LIN {X 0,Y 388.393,Z 704.087,A -85,B 0,C 180,E1 -23559.854,E2 -23559.854} C_VEL
LIN {X 0,Y 400.252,Z 573.446,A -85,B 0,C 180,E1 -23561.917,E2 -23561.917} C_VEL
LIN {X 0,Y 395.946,Z 563.972,A -85,B 0,C 180,E1 -23564.361,E2 -23564.361} C_VEL
LIN {X 0,Y 391.725,Z 556.337,A -85,B 0,C 180,E1 -23567.094,E2 -23567.094} C_VEL
LIN {X 0,Y 388.594,Z 550.898,A -85,B 0,C 180,E1 -23569.548,E2 -23569.548} C_VEL
LIN {X 0,Y 386.254,Z 546.876,A -85,B 0,C 180,E1 -23571.815,E2 -23571.815} C_VEL
LIN {X 0,Y 383.997,Z 542.829,A -85,B 0,C 180,E1 -23574.771,E2 -23574.771} C_VEL
LIN {X 0,Y 382.142,Z 538.278,A -85,B 0,C 180,E1 -23581.349,E2 -23581.349} C_VEL
LIN {X 0,Y 384.382,Z 543.419,A -85,B 0,C 180,E1 -23588.226,E2 -23588.226} C_VEL
LIN {X 0,Y 387.171,Z 548.383,A -85,B 0,C 180,E1 -23591.546,E2 -23591.546} C_VEL
LIN {X 0,Y 389.894,Z 553.166,A -85,B 0,C 180,E1 -23593.949,E2 -23593.949} C_VEL
LIN {X 0,Y 393.621,Z 559.599,A -85,B 0,C 180,E1 -23596.605,E2 -23596.605} C_VEL
LIN {X 0,Y 398.687,Z 569.021,A -85,B 0,C 180,E1 -23599.599,E2 -23599.599} C_VEL
LIN {X 0,Y 400.284,Z 572.367,A -85,B 0,C 180,E1 -23600.456,E2 -23600.456} C_VEL
LIN {X 0,Y 384.057,Z 748.302,A -85,B 0,C 180,E1 -23603.233,E2 -23603.233} C_VEL
LIN {X 0,Y 380.026,Z 774.745,A -85,B 0,C 180,E1 -23603.787,E2 -23603.787} C_VEL
LIN {X 0,Y 375.691,Z 795.491,A -85,B 0,C 180,E1 -23604.362,E2 -23604.362} C_VEL
LIN {X 0,Y 369.224,Z 820.189,A -85,B 0,C 180,E1 -23605.244,E2 -23605.244} C_VEL
LIN {X 0,Y 362.641,Z 840.771,A -85,B 0,C 180,E1 -23606.178,E2 -23606.178} C_VEL
LIN {X 0,Y 354.698,Z 862.408,A -85,B 0,C 180,E1 -23607.379,E2 -23607.379} C_VEL
LIN {X 0,Y 345.362,Z 883.966,A -85,B 0,C 180,E1 -23608.861,E2 -23608.861} C_VEL
LIN {X 0,Y 335.768,Z 903.879,A -85,B 0,C 180,E1 -23610.523,E2 -23610.523} C_VEL
LIN {X 0,Y 325.015,Z 923.613,A -85,B 0,C 180,E1 -23612.548,E2 -23612.548} C_VEL
LIN {X 0,Y 314.859,Z 940.708,A -85,B 0,C 180,E1 -23614.664,E2 -23614.664} C_VEL
LIN {X 0,Y 303.227,Z 958.602,A -85,B 0,C 180,E1 -23617.373,E2 -23617.373} C_VEL
LIN {X 0,Y 292.874,Z 973.436,A -85,B 0,C 180,E1 -23620.115,E2 -23620.115} C_VEL
LIN {X 0,Y 281.008,Z 989.437,A -85,B 0,C 180,E1 -23623.754,E2 -23623.754} C_VEL
LIN {X 0,Y 271.257,Z 1001.963,A -85,B 0,C 180,E1 -23627.293,E2 -23627.293} C_VEL
LIN {X 0,Y 261.14,Z 1014.647,A -85,B 0,C 180,E1 -23631.715,E2 -23631.715} C_VEL
LIN {X 0,Y 252.983,Z 1024.7,A -85,B 0,C 180,E1 -23636.132,E2 -23636.132} C_VEL
LIN {X 0,Y 245.579,Z 1034.158,A -85,B 0,C 180,E1 -23641.286,E2 -23641.286} C_VEL
LIN {X 0,Y 239.901,Z 1041.714,A -85,B 0,C 180,E1 -23646.675,E2 -23646.675} C_VEL
LIN {X 0,Y 235.924,Z 1047.812,A -85,B 0,C 180,E1 -23652.233,E2 -23652.233} C_VEL
LIN {X 0,Y 233.421,Z 1052.417,A -85,B 0,C 180,E1 -23658.135,E2 -23658.135} C_VEL
LIN {X 0,Y 232.411,Z 1055.085,A -85,B 0,C 180,E1 -23663.081,E2 -23663.081} C_VEL
LIN {X 0,Y 232.071,Z 1056.714,A -85,B 0,C 180,E1 -23668.025,E2 -23668.025} C_VEL
LIN {X 0,Y 232.018,Z 1057.307,A -85,B 0,C 180,E1 -23673.212,E2 -23673.212} C_VEL
LIN {X 0,Y 232.196,Z 1056.634,A -85,B 0,C 180,E1 -23678.419,E2 -23678.419} C_VEL
LIN {X 0,Y 232.853,Z 1054.948,A -85,B 0,C 180,E1 -23683.408,E2 -23683.408} C_VEL
LIN {X 0,Y 234.592,Z 1051.893,A -85,B 0,C 180,E1 -23688.901,E2 -23688.901} C_VEL
LIN {X 0,Y 238.088,Z 1046.847,A -85,B 0,C 180,E1 -23694.888,E2 -23694.888} C_VEL
LIN {X 0,Y 242.615,Z 1041.161,A -85,B 0,C 180,E1 -23699.913,E2 -23699.913} C_VEL
LIN {X 0,Y 250.02,Z 1032.531,A -85,B 0,C 180,E1 -23705.725,E2 -23705.725} C_VEL
LIN {X 0,Y 257.882,Z 1023.616,A -85,B 0,C 180,E1 -23710.354,E2 -23710.354} C_VEL
LIN {X 0,Y 268.413,Z 1011.672,A -85,B 0,C 180,E1 -23715.246,E2 -23715.246} C_VEL
LIN {X 0,Y 278.302,Z 1000.135,A -85,B 0,C 180,E1 -23718.981,E2 -23718.981} C_VEL
LIN {X 0,Y 290.19,Z 985.74,A -85,B 0,C 180,E1 -23722.744,E2 -23722.744} C_VEL
LIN {X 0,Y 301.246,Z 971.426,A -85,B 0,C 180,E1 -23725.739,E2 -23725.739} C_VEL
LIN {X 0,Y 313.044,Z 955.275,A -85,B 0,C 180,E1 -23728.52,E2 -23728.52} C_VEL
LIN {X 0,Y 324.773,Z 937.569,A -85,B 0,C 180,E1 -23730.969,E2 -23730.969} C_VEL
LIN {X 0,Y 335.952,Z 919.34,A -85,B 0,C 180,E1 -23733.049,E2 -23733.049} C_VEL
LIN {X 0,Y 346.746,Z 899.544,A -85,B 0,C 180,E1 -23734.886,E2 -23734.886} C_VEL
LIN {X 0,Y 355.593,Z 881.622,A -85,B 0,C 180,E1 -23736.264,E2 -23736.264} C_VEL
LIN {X 0,Y 365.537,Z 858.721,A -85,B 0,C 180,E1 -23737.71,E2 -23737.71} C_VEL
LIN {X 0,Y 372.878,Z 839.111,A -85,B 0,C 180,E1 -23738.723,E2 -23738.723} C_VEL
LIN {X 0,Y 380.335,Z 815.96,A -85,B 0,C 180,E1 -23739.694,E2 -23739.694} C_VEL
LIN {X 0,Y 386.25,Z 793.125,A -85,B 0,C 180,E1 -23740.44,E2 -23740.44} C_VEL
LIN {X 0,Y 391.244,Z 769.089,A -85,B 0,C 180,E1 -23741.046,E2 -23741.046} C_VEL
LIN {X 0,Y 394.683,Z 744.791,A -85,B 0,C 180,E1 -23741.5,E2 -23741.5} C_VEL
LIN {X 0,Y 410.348,Z 579.625,A -85,B 0,C 180,E1 -23744.054,E2 -23744.054} C_VEL
LIN {X 0,Y 405.942,Z 571.377,A -85,B 0,C 180,E1 -23746.83,E2 -23746.83} C_VEL
LIN {X 0,Y 402.359,Z 564.773,A -85,B 0,C 180,E1 -23749.621,E2 -23749.621} C_VEL
LIN {X 0,Y 400.956,Z 563.778,A -85,B 0,C 180,E1 -23750.779,E2 -23750.779} C_VEL
LIN {X 0,Y 397.256,Z 564.937,A -85,B 0,C 180,E1 -23754.266,E2 -23754.266} C_VEL
LIN {X 0,Y 396.971,Z 564.739,A -85,B 0,C 180,E1 -23754.666,E2 -23754.666} C_VEL
LIN {X 0,Y 395.189,Z 560.495,A -85,B 0,C 180,E1 -23760.87,E2 -23760.87} C_VEL
LIN {X 0,Y 397.102,Z 565.119,A -85,B 0,C 180,E1 -23767.233,E2 -23767.233} C_VEL
LIN {X 0,Y 399.583,Z 569.876,A -85,B 0,C 180,E1 -23770.38,E2 -23770.38} C_VEL
LIN {X 0,Y 402.269,Z 574.828,A -85,B 0,C 180,E1 -23772.854,E2 -23772.854} C_VEL
LIN {X 0,Y 405.294,Z 580.545,A -85,B 0,C 180,E1 -23775.123,E2 -23775.123} C_VEL
LIN {X 0,Y 407.597,Z 586.184,A -85,B 0,C 180,E1 -23776.699,E2 -23776.699} C_VEL
LIN {X 0,Y 391.12,Z 755.536,A -85,B 0,C 180,E1 -23779.285,E2 -23779.285} C_VEL
LIN {X 0,Y 386.856,Z 782.013,A -85,B 0,C 180,E1 -23779.789,E2 -23779.789} C_VEL
LIN {X 0,Y 382.071,Z 803.436,A -85,B 0,C 180,E1 -23780.299,E2 -23780.299} C_VEL
LIN {X 0,Y 375.038,Z 828.403,A -85,B 0,C 180,E1 -23781.071,E2 -23781.071} C_VEL
LIN {X 0,Y 367.984,Z 849.001,A -85,B 0,C 180,E1 -23781.886,E2 -23781.886} C_VEL
LIN {X 0,Y 359.022,Z 871.665,A -85,B 0,C 180,E1 -23783.007,E2 -23783.007} C_VEL
LIN {X 0,Y 349.433,Z 892.46,A -85,B 0,C 180,E1 -23784.304,E2 -23784.304} C_VEL
LIN {X 0,Y 338.891,Z 912.953,A -85,B 0,C 180,E1 -23785.856,E2 -23785.856} C_VEL
LIN {X 0,Y 327.505,Z 932.463,A -85,B 0,C 180,E1 -23787.701,E2 -23787.701} C_VEL
LIN {X 0,Y 316.516,Z 949.77,A -85,B 0,C 180,E1 -23789.687,E2 -23789.687} C_VEL
LIN {X 0,Y 303.867,Z 967.902,A -85,B 0,C 180,E1 -23792.256,E2 -23792.256} C_VEL
LIN {X 0,Y 293.193,Z 982.14,A -85,B 0,C 180,E1 -23794.725,E2 -23794.725} C_VEL
LIN {X 0,Y 280.683,Z 997.872,A -85,B 0,C 180,E1 -23798.068,E2 -23798.068} C_VEL
LIN {X 0,Y 269.384,Z 1011.222,A -85,B 0,C 180,E1 -23801.637,E2 -23801.637} C_VEL
LIN {X 0,Y 258.376,Z 1023.94,A -85,B 0,C 180,E1 -23805.847,E2 -23805.847} C_VEL
LIN {X 0,Y 248.504,Z 1034.966,A -85,B 0,C 180,E1 -23810.526,E2 -23810.526} C_VEL
LIN {X 0,Y 239.962,Z 1044.827,A -85,B 0,C 180,E1 -23815.769,E2 -23815.769} C_VEL
LIN {X 0,Y 233.287,Z 1052.746,A -85,B 0,C 180,E1 -23821.312,E2 -23821.312} C_VEL
LIN {X 0,Y 228.711,Z 1058.908,A -85,B 0,C 180,E1 -23826.83,E2 -23826.83} C_VEL
LIN {X 0,Y 225.515,Z 1064.125,A -85,B 0,C 180,E1 -23833.277,E2 -23833.277} C_VEL
LIN {X 0,Y 224.312,Z 1066.99,A -85,B 0,C 180,E1 -23838.428,E2 -23838.428} C_VEL
LIN {X 0,Y 223.979,Z 1068.777,A -85,B 0,C 180,E1 -23843.592,E2 -23843.592} C_VEL
LIN {X 0,Y 224.01,Z 1069.469,A -85,B 0,C 180,E1 -23848.721,E2 -23848.721} C_VEL
LIN {X 0,Y 223.991,Z 1069.015,A -85,B 0,C 180,E1 -23853.583,E2 -23853.583} C_VEL
LIN {X 0,Y 224.053,Z 1067.383,A -85,B 0,C 180,E1 -23858.727,E2 -23858.727} C_VEL
LIN {X 0,Y 224.71,Z 1064.64,A -85,B 0,C 180,E1 -23863.903,E2 -23863.903} C_VEL
LIN {X 0,Y 226.6,Z 1060.347,A -85,B 0,C 180,E1 -23869.594,E2 -23869.594} C_VEL
LIN {X 0,Y 230.424,Z 1053.913,A -85,B 0,C 180,E1 -23875.718,E2 -23875.718} C_VEL
LIN {X 0,Y 235.435,Z 1046.841,A -85,B 0,C 180,E1 -23880.923,E2 -23880.923} C_VEL
LIN {X 0,Y 243.47,Z 1036.499,A -85,B 0,C 180,E1 -23886.841,E2 -23886.841} C_VEL
LIN {X 0,Y 251.465,Z 1026.59,A -85,B 0,C 180,E1 -23891.304,E2 -23891.304} C_VEL
LIN {X 0,Y 262.304,Z 1013.248,A -85,B 0,C 180,E1 -23896.092,E2 -23896.092} C_VEL
LIN {X 0,Y 272.513,Z 1000.343,A -85,B 0,C 180,E1 -23899.776,E2 -23899.776} C_VEL
LIN {X 0,Y 284.845,Z 984.13,A -85,B 0,C 180,E1 -23903.5,E2 -23903.5} C_VEL
LIN {X 0,Y 295.676,Z 968.974,A -85,B 0,C 180,E1 -23906.294,E2 -23906.294} C_VEL
LIN {X 0,Y 307.858,Z 950.808,A -85,B 0,C 180,E1 -23909.031,E2 -23909.031} C_VEL
LIN {X 0,Y 318.866,Z 932.772,A -85,B 0,C 180,E1 -23911.217,E2 -23911.217} C_VEL
LIN {X 0,Y 329.909,Z 913.124,A -85,B 0,C 180,E1 -23913.179,E2 -23913.179} C_VEL
LIN {X 0,Y 340.246,Z 892.323,A -85,B 0,C 180,E1 -23914.84,E2 -23914.84} C_VEL
LIN {X 0,Y 349.638,Z 871.278,A -85,B 0,C 180,E1 -23916.224,E2 -23916.224} C_VEL
LIN {X 0,Y 358.028,Z 849.339,A -85,B 0,C 180,E1 -23917.37,E2 -23917.37} C_VEL
LIN {X 0,Y 364.543,Z 829.829,A -85,B 0,C 180,E1 -23918.195,E2 -23918.195} C_VEL
LIN {X 0,Y 371.552,Z 804.574,A -85,B 0,C 180,E1 -23919.038,E2 -23919.038} C_VEL
LIN {X 0,Y 376.275,Z 783.017,A -85,B 0,C 180,E1 -23919.588,E2 -23919.588} C_VEL
LIN {X 0,Y 380.395,Z 757.375,A -85,B 0,C 180,E1 -23920.106,E2 -23920.106} C_VEL
LIN {X 0,Y 387.874,Z 678.891,A -85,B 0,C 180,E1 -23921.359,E2 -23921.359} C_VEL
LIN {X 0,Y 397.206,Z 578.193,A -85,B 0,C 180,E1 -23922.946,E2 -23922.946} C_VEL
LIN {X 0,Y 393.989,Z 570.875,A -85,B 0,C 180,E1 -23924.884,E2 -23924.884} C_VEL
LIN {X 0,Y 389.653,Z 562.753,A -85,B 0,C 180,E1 -23927.853,E2 -23927.853} C_VEL
LIN {X 0,Y 387.019,Z 558.202,A -85,B 0,C 180,E1 -23930.032,E2 -23930.032} C_VEL
LIN {X 0,Y 384.996,Z 554.581,A -85,B 0,C 180,E1 -23932.088,E2 -23932.088} C_VEL
LIN {X 0,Y 382.923,Z 550.71,A -85,B 0,C 180,E1 -23934.907,E2 -23934.907} C_VEL
LIN {X 0,Y 381.159,Z 546.277,A -85,B 0,C 180,E1 -23941.353,E2 -23941.353} C_VEL
LIN {X 0,Y 383.252,Z 551.234,A -85,B 0,C 180,E1 -23948.024,E2 -23948.024} C_VEL
LIN {X 0,Y 385.89,Z 556.083,A -85,B 0,C 180,E1 -23951.282,E2 -23951.282} C_VEL
LIN {X 0,Y 388.626,Z 561.047,A -85,B 0,C 180,E1 -23953.768,E2 -23953.768} C_VEL
LIN {X 0,Y 392.071,Z 567.186,A -85,B 0,C 180,E1 -23956.292,E2 -23956.292} C_VEL
LIN {X 0,Y 397.023,Z 576.643,A -85,B 0,C 180,E1 -23959.302,E2 -23959.302} C_VEL
LIN {X 0,Y 397.249,Z 577.342,A -85,B 0,C 180,E1 -23959.442,E2 -23959.442} C_VEL
LIN {X 0,Y 381.103,Z 748.566,A -85,B 0,C 180,E1 -23962.119,E2 -23962.119} C_VEL
LIN {X 0,Y 377.011,Z 774.925,A -85,B 0,C 180,E1 -23962.664,E2 -23962.664} C_VEL
LIN {X 0,Y 372.563,Z 795.837,A -85,B 0,C 180,E1 -23963.234,E2 -23963.234} C_VEL
LIN {X 0,Y 365.89,Z 820.783,A -85,B 0,C 180,E1 -23964.113,E2 -23964.113} C_VEL
LIN {X 0,Y 359.2,Z 841.282,A -85,B 0,C 180,E1 -23965.032,E2 -23965.032} C_VEL
LIN {X 0,Y 350.7,Z 863.813,A -85,B 0,C 180,E1 -23966.275,E2 -23966.275} C_VEL
LIN {X 0,Y 341.559,Z 884.422,A -85,B 0,C 180,E1 -23967.681,E2 -23967.681} C_VEL
LIN {X 0,Y 331.921,Z 903.982,A -85,B 0,C 180,E1 -23969.297,E2 -23969.297} C_VEL
LIN {X 0,Y 320.748,Z 924.011,A -85,B 0,C 180,E1 -23971.333,E2 -23971.333} C_VEL
LIN {X 0,Y 310.371,Z 941.03,A -85,B 0,C 180,E1 -23973.429,E2 -23973.429} C_VEL
LIN {X 0,Y 298.317,Z 959.043,A -85,B 0,C 180,E1 -23976.151,E2 -23976.151} C_VEL
LIN {X 0,Y 287.709,Z 973.781,A -85,B 0,C 180,E1 -23978.879,E2 -23978.879} C_VEL
LIN {X 0,Y 275.441,Z 989.761,A -85,B 0,C 180,E1 -23982.53,E2 -23982.53} C_VEL
LIN {X 0,Y 265.709,Z 1001.804,A -85,B 0,C 180,E1 -23985.952,E2 -23985.952} C_VEL
LIN {X 0,Y 255.317,Z 1014.345,A -85,B 0,C 180,E1 -23990.331,E2 -23990.331} C_VEL
LIN {X 0,Y 246.25,Z 1024.988,A -85,B 0,C 180,E1 -23995.074,E2 -23995.074} C_VEL
LIN {X 0,Y 238.464,Z 1034.429,A -85,B 0,C 180,E1 -24000.345,E2 -24000.345} C_VEL
LIN {X 0,Y 232.457,Z 1041.978,A -85,B 0,C 180,E1 -24005.881,E2 -24005.881} C_VEL
LIN {X 0,Y 228.221,Z 1048.067,A -85,B 0,C 180,E1 -24011.612,E2 -24011.612} C_VEL
LIN {X 0,Y 225.534,Z 1052.657,A -85,B 0,C 180,E1 -24017.713,E2 -24017.713} C_VEL
LIN {X 0,Y 224.445,Z 1055.317,A -85,B 0,C 180,E1 -24022.834,E2 -24022.834} C_VEL
LIN {X 0,Y 224.076,Z 1056.938,A -85,B 0,C 180,E1 -24027.954,E2 -24027.954} C_VEL
LIN {X 0,Y 224.022,Z 1057.518,A -85,B 0,C 180,E1 -24033.326,E2 -24033.326} C_VEL
LIN {X 0,Y 224.227,Z 1056.838,A -85,B 0,C 180,E1 -24038.721,E2 -24038.721} C_VEL
LIN {X 0,Y 224.953,Z 1055.147,A -85,B 0,C 180,E1 -24043.888,E2 -24043.888} C_VEL
LIN {X 0,Y 226.857,Z 1052.087,A -85,B 0,C 180,E1 -24049.571,E2 -24049.571} C_VEL
LIN {X 0,Y 230.594,Z 1047.079,A -85,B 0,C 180,E1 -24055.697,E2 -24055.697} C_VEL
LIN {X 0,Y 235.517,Z 1041.292,A -85,B 0,C 180,E1 -24060.952,E2 -24060.952} C_VEL
LIN {X 0,Y 243.335,Z 1032.69,A -85,B 0,C 180,E1 -24066.865,E2 -24066.865} C_VEL
LIN {X 0,Y 251.188,Z 1024.22,A -85,B 0,C 180,E1 -24071.36,E2 -24071.36} C_VEL
LIN {X 0,Y 261.331,Z 1013.301,A -85,B 0,C 180,E1 -24075.998,E2 -24075.998} C_VEL
LIN {X 0,Y 271.895,Z 1001.438,A -85,B 0,C 180,E1 -24079.942,E2 -24079.942} C_VEL
LIN {X 0,Y 283.435,Z 988.076,A -85,B 0,C 180,E1 -24083.545,E2 -24083.545} C_VEL
LIN {X 0,Y 295.45,Z 973.104,A -85,B 0,C 180,E1 -24086.752,E2 -24086.752} C_VEL
LIN {X 0,Y 306.754,Z 958.132,A -85,B 0,C 180,E1 -24089.376,E2 -24089.376} C_VEL
LIN {X 0,Y 319.664,Z 939.475,A -85,B 0,C 180,E1 -24092.018,E2 -24092.018} C_VEL
LIN {X 0,Y 329.702,Z 923.628,A -85,B 0,C 180,E1 -24093.855,E2 -24093.855} C_VEL
LIN {X 0,Y 341.262,Z 903.562,A -85,B 0,C 180,E1 -24095.783,E2 -24095.783} C_VEL
LIN {X 0,Y 350.777,Z 884.924,A -85,B 0,C 180,E1 -24097.241,E2 -24097.241} C_VEL
LIN {X 0,Y 360.324,Z 864.084,A -85,B 0,C 180,E1 -24098.592,E2 -24098.592} C_VEL
LIN {X 0,Y 369.07,Z 841.614,A -85,B 0,C 180,E1 -24099.77,E2 -24099.77} C_VEL
LIN {X 0,Y 376.17,Z 820.468,A -85,B 0,C 180,E1 -24100.669,E2 -24100.669} C_VEL
LIN {X 0,Y 382.899,Z 795.872,A -85,B 0,C 180,E1 -24101.487,E2 -24101.487} C_VEL
LIN {X 0,Y 387.518,Z 774.707,A -85,B 0,C 180,E1 -24102.031,E2 -24102.031} C_VEL
LIN {X 0,Y 391.73,Z 747.973,A -85,B 0,C 180,E1 -24102.553,E2 -24102.553} C_VEL
LIN {X 0,Y 407.604,Z 585.037,A -85,B 0,C 180,E1 -24105.035,E2 -24105.035} C_VEL
LIN {X 0,Y 403.504,Z 577.084,A -85,B 0,C 180,E1 -24107.841,E2 -24107.841} C_VEL
LIN {X 0,Y 400.575,Z 571.719,A -85,B 0,C 180,E1 -24110.3,E2 -24110.3} C_VEL
LIN {X 0,Y 398.739,Z 568.31,A -85,B 0,C 180,E1 -24112.217,E2 -24112.217} C_VEL
LIN {X 0,Y 396.971,Z 564.739,A -85,B 0,C 180,E1 -24114.666,E2 -24114.666} C_VEL
LIN {X 0,Y 396.187,Z 564.939,A -85,B 0,C 180,E1 -24115.781,E2 -24115.781} C_VEL
LIN {X 0,Y 394.357,Z 569.171,A -85,B 0,C 180,E1 -24118.868,E2 -24118.868} C_VEL
LIN {X 0,Y 394.191,Z 569.196,A -85,B 0,C 180,E1 -24119.755,E2 -24119.755} C_VEL
LIN {X 0,Y 394.201,Z 568.561,A -85,B 0,C 180,E1 -24121.017,E2 -24121.017} C_VEL
LIN {X 0,Y 395.985,Z 572.93,A -85,B 0,C 180,E1 -24127.034,E2 -24127.034} C_VEL
LIN {X 0,Y 398.325,Z 577.571,A -85,B 0,C 180,E1 -24130.12,E2 -24130.12} C_VEL
LIN {X 0,Y 400.85,Z 582.375,A -85,B 0,C 180,E1 -24132.534,E2 -24132.534} C_VEL
LIN {X 0,Y 403.733,Z 588.041,A -85,B 0,C 180,E1 -24134.779,E2 -24134.779} C_VEL
LIN {X 0,Y 404.955,Z 591.394,A -85,B 0,C 180,E1 -24135.686,E2 -24135.686} C_VEL
LIN {X 0,Y 388.666,Z 755.37,A -85,B 0,C 180,E1 -24138.162,E2 -24138.162} C_VEL
LIN {X 0,Y 384.319,Z 781.902,A -85,B 0,C 180,E1 -24138.657,E2 -24138.657} C_VEL
LIN {X 0,Y 379.456,Z 803.341,A -85,B 0,C 180,E1 -24139.156,E2 -24139.156} C_VEL
LIN {X 0,Y 372.227,Z 828.54,A -85,B 0,C 180,E1 -24139.918,E2 -24139.918} C_VEL
LIN {X 0,Y 365.063,Z 849.096,A -85,B 0,C 180,E1 -24140.715,E2 -24140.715} C_VEL
LIN {X 0,Y 355.947,Z 871.697,A -85,B 0,C 180,E1 -24141.812,E2 -24141.812} C_VEL
LIN {X 0,Y 346.182,Z 892.468,A -85,B 0,C 180,E1 -24143.083,E2 -24143.083} C_VEL
LIN {X 0,Y 335.432,Z 912.933,A -85,B 0,C 180,E1 -24144.608,E2 -24144.608} C_VEL
LIN {X 0,Y 323.799,Z 932.413,A -85,B 0,C 180,E1 -24146.425,E2 -24146.425} C_VEL
LIN {X 0,Y 312.182,Z 950.261,A -85,B 0,C 180,E1 -24148.454,E2 -24148.454} C_VEL
LIN {X 0,Y 299.551,Z 967.837,A -85,B 0,C 180,E1 -24150.934,E2 -24150.934} C_VEL
LIN {X 0,Y 288.164,Z 982.576,A -85,B 0,C 180,E1 -24153.484,E2 -24153.484} C_VEL
LIN {X 0,Y 274.431,Z 999.159,A -85,B 0,C 180,E1 -24157.067,E2 -24157.067} C_VEL
LIN {X 0,Y 263.197,Z 1011.954,A -85,B 0,C 180,E1 -24160.553,E2 -24160.553} C_VEL
LIN {X 0,Y 250.983,Z 1025.361,A -85,B 0,C 180,E1 -24165.165,E2 -24165.165} C_VEL
LIN {X 0,Y 241.502,Z 1035.524,A -85,B 0,C 180,E1 -24169.625,E2 -24169.625} C_VEL
LIN {X 0,Y 232.464,Z 1045.385,A -85,B 0,C 180,E1 -24175.105,E2 -24175.105} C_VEL
LIN {X 0,Y 225.807,Z 1052.876,A -85,B 0,C 180,E1 -24180.56,E2 -24180.56} C_VEL
LIN {X 0,Y 220.639,Z 1059.497,A -85,B 0,C 180,E1 -24186.78,E2 -24186.78} C_VEL
LIN {X 0,Y 217.522,Z 1064.242,A -85,B 0,C 180,E1 -24193.166,E2 -24193.166} C_VEL
LIN {X 0,Y 216.293,Z 1067.025,A -85,B 0,C 180,E1 -24198.536,E2 -24198.536} C_VEL
LIN {X 0,Y 215.98,Z 1068.863,A -85,B 0,C 180,E1 -24204.478,E2 -24204.478} C_VEL
LIN {X 0,Y 216.025,Z 1069.208,A -85,B 0,C 180,E1 -24209.735,E2 -24209.735} C_VEL
LIN {X 0,Y 215.988,Z 1068.582,A -85,B 0,C 180,E1 -24214.514,E2 -24214.514} C_VEL
LIN {X 0,Y 216.102,Z 1066.917,A -85,B 0,C 180,E1 -24219.588,E2 -24219.588} C_VEL
LIN {X 0,Y 216.871,Z 1064.236,A -85,B 0,C 180,E1 -24224.689,E2 -24224.689} C_VEL
LIN {X 0,Y 219.153,Z 1059.671,A -85,B 0,C 180,E1 -24230.847,E2 -24230.847} C_VEL
LIN {X 0,Y 223.315,Z 1053.221,A -85,B 0,C 180,E1 -24236.998,E2 -24236.998} C_VEL
LIN {X 0,Y 229.108,Z 1045.667,A -85,B 0,C 180,E1 -24242.615,E2 -24242.615} C_VEL
LIN {X 0,Y 237.26,Z 1035.745,A -85,B 0,C 180,E1 -24248.28,E2 -24248.28} C_VEL
LIN {X 0,Y 245.743,Z 1025.772,A -85,B 0,C 180,E1 -24252.804,E2 -24252.804} C_VEL
LIN {X 0,Y 257.141,Z 1012.292,A -85,B 0,C 180,E1 -24257.63,E2 -24257.63} C_VEL
LIN {X 0,Y 267.758,Z 999.38,A -85,B 0,C 180,E1 -24261.303,E2 -24261.303} C_VEL
LIN {X 0,Y 280.637,Z 982.934,A -85,B 0,C 180,E1 -24265.032,E2 -24265.032} C_VEL
LIN {X 0,Y 291.856,Z 967.687,A -85,B 0,C 180,E1 -24267.802,E2 -24267.802} C_VEL
LIN {X 0,Y 305.139,Z 948.186,A -85,B 0,C 180,E1 -24270.649,E2 -24270.649} C_VEL
LIN {X 0,Y 315.369,Z 931.769,A -85,B 0,C 180,E1 -24272.592,E2 -24272.592} C_VEL
LIN {X 0,Y 327.106,Z 911.145,A -85,B 0,C 180,E1 -24274.592,E2 -24274.592} C_VEL
LIN {X 0,Y 336.859,Z 891.881,A -85,B 0,C 180,E1 -24276.096,E2 -24276.096} C_VEL
LIN {X 0,Y 346.84,Z 869.832,A -85,B 0,C 180,E1 -24277.511,E2 -24277.511} C_VEL
LIN {X 0,Y 355.392,Z 847.669,A -85,B 0,C 180,E1 -24278.632,E2 -24278.632} C_VEL
LIN {X 0,Y 363.074,Z 824.71,A -85,B 0,C 180,E1 -24279.559,E2 -24279.559} C_VEL
LIN {X 0,Y 369.397,Z 801.15,A -85,B 0,C 180,E1 -24280.285,E2 -24280.285} C_VEL
LIN {X 0,Y 374.38,Z 778.046,A -85,B 0,C 180,E1 -24280.841,E2 -24280.841} C_VEL
LIN {X 0,Y 378.077,Z 753.063,A -85,B 0,C 180,E1 -24281.314,E2 -24281.314} C_VEL
LIN {X 0,Y 394.351,Z 583.045,A -85,B 0,C 180,E1 -24283.956,E2 -24283.956} C_VEL
LIN {X 0,Y 391.902,Z 577.444,A -85,B 0,C 180,E1 -24285.52,E2 -24285.52} C_VEL
LIN {X 0,Y 387.716,Z 569.519,A -85,B 0,C 180,E1 -24288.546,E2 -24288.546} C_VEL
LIN {X 0,Y 385.551,Z 565.623,A -85,B 0,C 180,E1 -24290.446,E2 -24290.446} C_VEL
LIN {X 0,Y 383.879,Z 562.467,A -85,B 0,C 180,E1 -24292.216,E2 -24292.216} C_VEL
LIN {X 0,Y 381.85,Z 558.59,A -85,B 0,C 180,E1 -24295.043,E2 -24295.043} C_VEL
LIN {X 0,Y 380.177,Z 554.278,A -85,B 0,C 180,E1 -24301.356,E2 -24301.356} C_VEL
LIN {X 0,Y 382.169,Z 559.167,A -85,B 0,C 180,E1 -24307.895,E2 -24307.895} C_VEL
LIN {X 0,Y 384.686,Z 563.928,A -85,B 0,C 180,E1 -24311.09,E2 -24311.09} C_VEL
LIN {X 0,Y 387.275,Z 568.76,A -85,B 0,C 180,E1 -24313.513,E2 -24313.513} C_VEL
LIN {X 0,Y 390.585,Z 574.877,A -85,B 0,C 180,E1 -24316.012,E2 -24316.012} C_VEL
LIN {X 0,Y 394.342,Z 582.297,A -85,B 0,C 180,E1 -24318.412,E2 -24318.412} C_VEL
LIN {X 0,Y 378.296,Z 748.83,A -85,B 0,C 180,E1 -24320.989,E2 -24320.989} C_VEL
LIN {X 0,Y 374.118,Z 775.234,A -85,B 0,C 180,E1 -24321.526,E2 -24321.526} C_VEL
LIN {X 0,Y 369.59,Z 796.141,A -85,B 0,C 180,E1 -24322.086,E2 -24322.086} C_VEL
LIN {X 0,Y 363.105,Z 820.101,A -85,B 0,C 180,E1 -24322.91,E2 -24322.91} C_VEL
LIN {X 0,Y 356.291,Z 840.703,A -85,B 0,C 180,E1 -24323.811,E2 -24323.811} C_VEL
LIN {X 0,Y 347.935,Z 862.643,A -85,B 0,C 180,E1 -24324.989,E2 -24324.989} C_VEL
LIN {X 0,Y 338.291,Z 884.075,A -85,B 0,C 180,E1 -24326.417,E2 -24326.417} C_VEL
LIN {X 0,Y 328.842,Z 902.891,A -85,B 0,C 180,E1 -24327.938,E2 -24327.938} C_VEL
LIN {X 0,Y 317.357,Z 923.205,A -85,B 0,C 180,E1 -24329.953,E2 -24329.953} C_VEL
LIN {X 0,Y 307.054,Z 939.742,A -85,B 0,C 180,E1 -24331.946,E2 -24331.946} C_VEL
LIN {X 0,Y 294.341,Z 958.4,A -85,B 0,C 180,E1 -24334.706,E2 -24334.706} C_VEL
LIN {X 0,Y 283.827,Z 972.616,A -85,B 0,C 180,E1 -24337.297,E2 -24337.297} C_VEL
LIN {X 0,Y 271.761,Z 988.016,A -85,B 0,C 180,E1 -24340.718,E2 -24340.718} C_VEL
LIN {X 0,Y 260.571,Z 1001.343,A -85,B 0,C 180,E1 -24344.46,E2 -24344.46} C_VEL
LIN {X 0,Y 249.83,Z 1013.835,A -85,B 0,C 180,E1 -24348.802,E2 -24348.802} C_VEL
LIN {X 0,Y 240.003,Z 1024.826,A -85,B 0,C 180,E1 -24353.73,E2 -24353.73} C_VEL
LIN {X 0,Y 231.738,Z 1034.345,A -85,B 0,C 180,E1 -24359.106,E2 -24359.106} C_VEL
LIN {X 0,Y 225.118,Z 1042.167,A -85,B 0,C 180,E1 -24364.972,E2 -24364.972} C_VEL
LIN {X 0,Y 220.545,Z 1048.322,A -85,B 0,C 180,E1 -24370.948,E2 -24370.948} C_VEL
LIN {X 0,Y 217.661,Z 1052.896,A -85,B 0,C 180,E1 -24377.262,E2 -24377.262} C_VEL
LIN {X 0,Y 216.482,Z 1055.548,A -85,B 0,C 180,E1 -24382.569,E2 -24382.569} C_VEL
LIN {X 0,Y 216.081,Z 1057.161,A -85,B 0,C 180,E1 -24387.879,E2 -24387.879} C_VEL
LIN {X 0,Y 216.023,Z 1057.746,A -85,B 0,C 180,E1 -24393.184,E2 -24393.184} C_VEL
LIN {X 0,Y 216.234,Z 1057.109,A -85,B 0,C 180,E1 -24398.777,E2 -24398.777} C_VEL
LIN {X 0,Y 217.003,Z 1055.456,A -85,B 0,C 180,E1 -24404.135,E2 -24404.135} C_VEL
LIN {X 0,Y 218.92,Z 1052.565,A -85,B 0,C 180,E1 -24409.799,E2 -24409.799} C_VEL
LIN {X 0,Y 222.985,Z 1047.508,A -85,B 0,C 180,E1 -24416.355,E2 -24416.355} C_VEL
LIN {X 0,Y 228.181,Z 1041.755,A -85,B 0,C 180,E1 -24421.776,E2 -24421.776} C_VEL
LIN {X 0,Y 236.021,Z 1033.63,A -85,B 0,C 180,E1 -24427.607,E2 -24427.607} C_VEL
LIN {X 0,Y 244.575,Z 1024.825,A -85,B 0,C 180,E1 -24432.42,E2 -24432.42} C_VEL
LIN {X 0,Y 255.125,Z 1013.998,A -85,B 0,C 180,E1 -24437.13,E2 -24437.13} C_VEL
LIN {X 0,Y 266.567,Z 1001.642,A -85,B 0,C 180,E1 -24441.279,E2 -24441.279} C_VEL
LIN {X 0,Y 278.914,Z 987.844,A -85,B 0,C 180,E1 -24444.999,E2 -24444.999} C_VEL
LIN {X 0,Y 291.601,Z 972.449,A -85,B 0,C 180,E1 -24448.253,E2 -24448.253} C_VEL
LIN {X 0,Y 304.417,Z 955.9,A -85,B 0,C 180,E1 -24451.086,E2 -24451.086} C_VEL
LIN {X 0,Y 316.764,Z 938.223,A -85,B 0,C 180,E1 -24453.494,E2 -24453.494} C_VEL
LIN {X 0,Y 328.092,Z 920.623,A -85,B 0,C 180,E1 -24455.465,E2 -24455.465} C_VEL
LIN {X 0,Y 339.836,Z 900.107,A -85,B 0,C 180,E1 -24457.329,E2 -24457.329} C_VEL
LIN {X 0,Y 349.323,Z 881.65,A -85,B 0,C 180,E1 -24458.701,E2 -24458.701} C_VEL
LIN {X 0,Y 359.482,Z 859.074,A -85,B 0,C 180,E1 -24460.075,E2 -24460.075} C_VEL
LIN {X 0,Y 366.898,Z 840.001,A -85,B 0,C 180,E1 -24461.025,E2 -24461.025} C_VEL
LIN {X 0,Y 374.661,Z 816.827,A -85,B 0,C 180,E1 -24461.966,E2 -24461.966} C_VEL
LIN {X 0,Y 380.859,Z 793.719,A -85,B 0,C 180,E1 -24462.693,E2 -24462.693} C_VEL
LIN {X 0,Y 386.033,Z 769.656,A -85,B 0,C 180,E1 -24463.277,E2 -24463.277} C_VEL
LIN {X 0,Y 389.616,Z 745.218,A -85,B 0,C 180,E1 -24463.718,E2 -24463.718} C_VEL
LIN {X 0,Y 404.922,Z 590.346,A -85,B 0,C 180,E1 -24466.068,E2 -24466.068} C_VEL
LIN {X 0,Y 401.251,Z 583.168,A -85,B 0,C 180,E1 -24468.792,E2 -24468.792} C_VEL
LIN {X 0,Y 398.992,Z 578.889,A -85,B 0,C 180,E1 -24470.843,E2 -24470.843} C_VEL
LIN {X 0,Y 397.505,Z 576.015,A -85,B 0,C 180,E1 -24472.484,E2 -24472.484} C_VEL
LIN {X 0,Y 395.726,Z 572.441,A -85,B 0,C 180,E1 -24475.072,E2 -24475.072} C_VEL
LIN {X 0,Y 394.191,Z 569.196,A -85,B 0,C 180,E1 -24479.755,E2 -24479.755} C_VEL
LIN {X 0,Y 394.072,Z 569.689,A -85,B 0,C 180,E1 -24480.392,E2 -24480.392} C_VEL
LIN {X 0,Y 393.674,Z 572.986,A -85,B 0,C 180,E1 -24481.377,E2 -24481.377} C_VEL
LIN {X 0,Y 393.316,Z 577.058,A -85,B 0,C 180,E1 -24482.464,E2 -24482.464} C_VEL
LIN {X 0,Y 393.327,Z 577.972,A -85,B 0,C 180,E1 -24483.003,E2 -24483.003} C_VEL
LIN {X 0,Y 394.911,Z 580.859,A -85,B 0,C 180,E1 -24486.908,E2 -24486.908} C_VEL
LIN {X 0,Y 397.137,Z 585.407,A -85,B 0,C 180,E1 -24489.931,E2 -24489.931} C_VEL
LIN {X 0,Y 399.686,Z 590.391,A -85,B 0,C 180,E1 -24492.424,E2 -24492.424} C_VEL
LIN {X 0,Y 402.368,Z 595.995,A -85,B 0,C 180,E1 -24494.573,E2 -24494.573} C_VEL
LIN {X 0,Y 402.437,Z 596.658,A -85,B 0,C 180,E1 -24494.661,E2 -24494.661} C_VEL
LIN {X 0,Y 386.359,Z 755.249,A -85,B 0,C 180,E1 -24497.025,E2 -24497.025} C_VEL
LIN {X 0,Y 381.94,Z 781.772,A -85,B 0,C 180,E1 -24497.511,E2 -24497.511} C_VEL
LIN {X 0,Y 377,Z 803.226,A -85,B 0,C 180,E1 -24497.997,E2 -24497.997} C_VEL
LIN {X 0,Y 369.57,Z 828.679,A -85,B 0,C 180,E1 -24498.748,E2 -24498.748} C_VEL
LIN {X 0,Y 362.338,Z 849.079,A -85,B 0,C 180,E1 -24499.52,E2 -24499.52} C_VEL
LIN {X 0,Y 352.609,Z 872.629,A -85,B 0,C 180,E1 -24500.646,E2 -24500.646} C_VEL
LIN {X 0,Y 343.092,Z 892.475,A -85,B 0,C 180,E1 -24501.841,E2 -24501.841} C_VEL
LIN {X 0,Y 332.136,Z 912.908,A -85,B 0,C 180,E1 -24503.336,E2 -24503.336} C_VEL
LIN {X 0,Y 320.172,Z 932.497,A -85,B 0,C 180,E1 -24505.133,E2 -24505.133} C_VEL
LIN {X 0,Y 307.996,Z 950.753,A -85,B 0,C 180,E1 -24507.187,E2 -24507.187} C_VEL
LIN {X 0,Y 294.932,Z 968.373,A -85,B 0,C 180,E1 -24509.668,E2 -24509.668} C_VEL
LIN {X 0,Y 283.199,Z 983.106,A -85,B 0,C 180,E1 -24512.218,E2 -24512.218} C_VEL
LIN {X 0,Y 269.54,Z 999.036,A -85,B 0,C 180,E1 -24515.668,E2 -24515.668} C_VEL
LIN {X 0,Y 258.487,Z 1011.181,A -85,B 0,C 180,E1 -24518.966,E2 -24518.966} C_VEL
LIN {X 0,Y 246.232,Z 1024.161,A -85,B 0,C 180,E1 -24523.375,E2 -24523.375} C_VEL
LIN {X 0,Y 235.946,Z 1034.651,A -85,B 0,C 180,E1 -24527.966,E2 -24527.966} C_VEL
LIN {X 0,Y 226.454,Z 1044.49,A -85,B 0,C 180,E1 -24533.41,E2 -24533.41} C_VEL
LIN {X 0,Y 218.925,Z 1052.388,A -85,B 0,C 180,E1 -24539.234,E2 -24539.234} C_VEL
LIN {X 0,Y 213.517,Z 1058.736,A -85,B 0,C 180,E1 -24545.298,E2 -24545.298} C_VEL
LIN {X 0,Y 209.917,Z 1063.715,A -85,B 0,C 180,E1 -24551.964,E2 -24551.964} C_VEL
LIN {X 0,Y 208.437,Z 1066.587,A -85,B 0,C 180,E1 -24557.533,E2 -24557.533} C_VEL
LIN {X 0,Y 207.988,Z 1068.365,A -85,B 0,C 180,E1 -24563.097,E2 -24563.097} C_VEL
LIN {X 0,Y 208.013,Z 1069.047,A -85,B 0,C 180,E1 -24568.623,E2 -24568.623} C_VEL
LIN {X 0,Y 207.992,Z 1068.569,A -85,B 0,C 180,E1 -24573.859,E2 -24573.859} C_VEL
LIN {X 0,Y 208.09,Z 1066.922,A -85,B 0,C 180,E1 -24579.403,E2 -24579.403} C_VEL
LIN {X 0,Y 208.923,Z 1064.162,A -85,B 0,C 180,E1 -24584.977,E2 -24584.977} C_VEL
LIN {X 0,Y 211.253,Z 1059.78,A -85,B 0,C 180,E1 -24591.182,E2 -24591.182} C_VEL
LIN {X 0,Y 215.751,Z 1053.27,A -85,B 0,C 180,E1 -24597.726,E2 -24597.726} C_VEL
LIN {X 0,Y 221.374,Z 1046.302,A -85,B 0,C 180,E1 -24603.129,E2 -24603.129} C_VEL
LIN {X 0,Y 230.388,Z 1035.929,A -85,B 0,C 180,E1 -24609.319,E2 -24609.319} C_VEL
LIN {X 0,Y 239.234,Z 1026.005,A -85,B 0,C 180,E1 -24613.932,E2 -24613.932} C_VEL
LIN {X 0,Y 251.067,Z 1012.628,A -85,B 0,C 180,E1 -24618.825,E2 -24618.825} C_VEL
LIN {X 0,Y 261.443,Z 1000.486,A -85,B 0,C 180,E1 -24622.342,E2 -24622.342} C_VEL
LIN {X 0,Y 274.013,Z 985.169,A -85,B 0,C 180,E1 -24625.928,E2 -24625.928} C_VEL
LIN {X 0,Y 286.148,Z 969.215,A -85,B 0,C 180,E1 -24628.882,E2 -24628.882} C_VEL
LIN {X 0,Y 298.699,Z 951.636,A -85,B 0,C 180,E1 -24631.526,E2 -24631.526} C_VEL
LIN {X 0,Y 310.577,Z 933.16,A -85,B 0,C 180,E1 -24633.74,E2 -24633.74} C_VEL
LIN {X 0,Y 322.111,Z 913.631,A -85,B 0,C 180,E1 -24635.655,E2 -24635.655} C_VEL
LIN {X 0,Y 332.832,Z 893.076,A -85,B 0,C 180,E1 -24637.262,E2 -24637.262} C_VEL
LIN {X 0,Y 342.167,Z 873.069,A -85,B 0,C 180,E1 -24638.549,E2 -24638.549} C_VEL
LIN {X 0,Y 351.268,Z 850.561,A -85,B 0,C 180,E1 -24639.706,E2 -24639.706} C_VEL
LIN {X 0,Y 358.058,Z 831.09,A -85,B 0,C 180,E1 -24640.507,E2 -24640.507} C_VEL
LIN {X 0,Y 365.017,Z 807.553,A -85,B 0,C 180,E1 -24641.282,E2 -24641.282} C_VEL
LIN {X 0,Y 370.365,Z 784.322,A -85,B 0,C 180,E1 -24641.862,E2 -24641.862} C_VEL
LIN {X 0,Y 374.65,Z 759.685,A -85,B 0,C 180,E1 -24642.354,E2 -24642.354} C_VEL
LIN {X 0,Y 379.883,Z 708.542,A -85,B 0,C 180,E1 -24643.164,E2 -24643.164} C_VEL
LIN {X 0,Y 391.56,Z 587.862,A -85,B 0,C 180,E1 -24645.013,E2 -24645.013} C_VEL
LIN {X 0,Y 388.687,Z 581.723,A -85,B 0,C 180,E1 -24646.992,E2 -24646.992} C_VEL
LIN {X 0,Y 384.958,Z 574.441,A -85,B 0,C 180,E1 -24650.054,E2 -24650.054} C_VEL
LIN {X 0,Y 382.634,Z 570.172,A -85,B 0,C 180,E1 -24652.492,E2 -24652.492} C_VEL
LIN {X 0,Y 380.687,Z 566.377,A -85,B 0,C 180,E1 -24655.33,E2 -24655.33} C_VEL
LIN {X 0,Y 379.195,Z 562.276,A -85,B 0,C 180,E1 -24661.36,E2 -24661.36} C_VEL
LIN {X 0,Y 381.047,Z 566.98,A -85,B 0,C 180,E1 -24667.691,E2 -24667.691} C_VEL
LIN {X 0,Y 383.419,Z 571.626,A -85,B 0,C 180,E1 -24670.822,E2 -24670.822} C_VEL
LIN {X 0,Y 385.933,Z 576.471,A -85,B 0,C 180,E1 -24673.255,E2 -24673.255} C_VEL
LIN {X 0,Y 389.259,Z 582.878,A -85,B 0,C 180,E1 -24675.838,E2 -24675.838} C_VEL
LIN {X 0,Y 391.526,Z 587.637,A -85,B 0,C 180,E1 -24677.372,E2 -24677.372} C_VEL
LIN {X 0,Y 375.637,Z 749.094,A -85,B 0,C 180,E1 -24679.842,E2 -24679.842} C_VEL
LIN {X 0,Y 371.401,Z 775.414,A -85,B 0,C 180,E1 -24680.368,E2 -24680.368} C_VEL
LIN {X 0,Y 366.788,Z 796.366,A -85,B 0,C 180,E1 -24680.917,E2 -24680.917} C_VEL
LIN {X 0,Y 360.072,Z 820.693,A -85,B 0,C 180,E1 -24681.74,E2 -24681.74} C_VEL
LIN {X 0,Y 353.14,Z 841.25,A -85,B 0,C 180,E1 -24682.625,E2 -24682.625} C_VEL
LIN {X 0,Y 344.606,Z 863.202,A -85,B 0,C 180,E1 -24683.786,E2 -24683.786} C_VEL
LIN {X 0,Y 334.798,Z 884.529,A -85,B 0,C 180,E1 -24685.187,E2 -24685.187} C_VEL
LIN {X 0,Y 324.731,Z 904.123,A -85,B 0,C 180,E1 -24686.754,E2 -24686.754} C_VEL
LIN {X 0,Y 313.167,Z 923.993,A -85,B 0,C 180,E1 -24688.718,E2 -24688.718} C_VEL
LIN {X 0,Y 302.44,Z 940.759,A -85,B 0,C 180,E1 -24690.731,E2 -24690.731} C_VEL
LIN {X 0,Y 289.803,Z 958.756,A -85,B 0,C 180,E1 -24693.389,E2 -24693.389} C_VEL
LIN {X 0,Y 278.691,Z 973.331,A -85,B 0,C 180,E1 -24696.044,E2 -24696.044} C_VEL
LIN {X 0,Y 266.527,Z 988.339,A -85,B 0,C 180,E1 -24699.392,E2 -24699.392} C_VEL
LIN {X 0,Y 254.93,Z 1001.657,A -85,B 0,C 180,E1 -24703.153,E2 -24703.153} C_VEL
LIN {X 0,Y 243.96,Z 1013.904,A -85,B 0,C 180,E1 -24707.448,E2 -24707.448} C_VEL
LIN {X 0,Y 233.898,Z 1024.664,A -85,B 0,C 180,E1 -24712.316,E2 -24712.316} C_VEL
LIN {X 0,Y 225.465,Z 1033.834,A -85,B 0,C 180,E1 -24717.547,E2 -24717.547} C_VEL
LIN {X 0,Y 218.219,Z 1041.913,A -85,B 0,C 180,E1 -24723.611,E2 -24723.611} C_VEL
LIN {X 0,Y 213.595,Z 1047.586,A -85,B 0,C 180,E1 -24729.159,E2 -24729.159} C_VEL
LIN {X 0,Y 209.997,Z 1052.826,A -85,B 0,C 180,E1 -24736.227,E2 -24736.227} C_VEL
LIN {X 0,Y 208.607,Z 1055.559,A -85,B 0,C 180,E1 -24741.733,E2 -24741.733} C_VEL
LIN {X 0,Y 208.115,Z 1057.186,A -85,B 0,C 180,E1 -24746.971,E2 -24746.971} C_VEL
LIN {X 0,Y 208.016,Z 1057.88,A -85,B 0,C 180,E1 -24752.204,E2 -24752.204} C_VEL
LIN {X 0,Y 208.182,Z 1057.575,A -85,B 0,C 180,E1 -24758.007,E2 -24758.007} C_VEL
LIN {X 0,Y 208.993,Z 1055.875,A -85,B 0,C 180,E1 -24764.123,E2 -24764.123} C_VEL
LIN {X 0,Y 210.945,Z 1053.094,A -85,B 0,C 180,E1 -24769.955,E2 -24769.955} C_VEL
LIN {X 0,Y 215.281,Z 1048.082,A -85,B 0,C 180,E1 -24776.904,E2 -24776.904} C_VEL
LIN {X 0,Y 220.897,Z 1042.216,A -85,B 0,C 180,E1 -24782.655,E2 -24782.655} C_VEL
LIN {X 0,Y 229.132,Z 1034.175,A -85,B 0,C 180,E1 -24788.636,E2 -24788.636} C_VEL
LIN {X 0,Y 238.514,Z 1024.975,A -85,B 0,C 180,E1 -24793.765,E2 -24793.765} C_VEL
LIN {X 0,Y 249.555,Z 1014.133,A -85,B 0,C 180,E1 -24798.525,E2 -24798.525} C_VEL
LIN {X 0,Y 261.467,Z 1001.766,A -85,B 0,C 180,E1 -24802.695,E2 -24802.695} C_VEL
LIN {X 0,Y 273.934,Z 988.303,A -85,B 0,C 180,E1 -24806.328,E2 -24806.328} C_VEL
LIN {X 0,Y 286.656,Z 973.382,A -85,B 0,C 180,E1 -24809.493,E2 -24809.493} C_VEL
LIN {X 0,Y 298.705,Z 958.289,A -85,B 0,C 180,E1 -24812.094,E2 -24812.094} C_VEL
LIN {X 0,Y 312.054,Z 939.937,A -85,B 0,C 180,E1 -24814.634,E2 -24814.634} C_VEL
LIN {X 0,Y 323.215,Z 923.089,A -85,B 0,C 180,E1 -24816.527,E2 -24816.527} C_VEL
LIN {X 0,Y 335.885,Z 901.738,A -85,B 0,C 180,E1 -24818.478,E2 -24818.478} C_VEL
LIN {X 0,Y 345.221,Z 884.06,A -85,B 0,C 180,E1 -24819.789,E2 -24819.789} C_VEL
LIN {X 0,Y 355.441,Z 862.284,A -85,B 0,C 180,E1 -24821.125,E2 -24821.125} C_VEL
LIN {X 0,Y 363.501,Z 842.146,A -85,B 0,C 180,E1 -24822.129,E2 -24822.129} C_VEL
LIN {X 0,Y 371.132,Z 820.134,A -85,B 0,C 180,E1 -24823.024,E2 -24823.024} C_VEL
LIN {X 0,Y 377.943,Z 795.836,A -85,B 0,C 180,E1 -24823.793,E2 -24823.793} C_VEL
LIN {X 0,Y 382.796,Z 774.16,A -85,B 0,C 180,E1 -24824.321,E2 -24824.321} C_VEL
LIN {X 0,Y 386.985,Z 748.089,A -85,B 0,C 180,E1 -24824.807,E2 -24824.807} C_VEL
LIN {X 0,Y 402.406,Z 595.907,A -85,B 0,C 180,E1 -24827.078,E2 -24827.078} C_VEL
LIN {X 0,Y 399.341,Z 589.769,A -85,B 0,C 180,E1 -24829.541,E2 -24829.541} C_VEL
LIN {X 0,Y 396.711,Z 584.355,A -85,B 0,C 180,E1 -24832.25,E2 -24832.25} C_VEL
LIN {X 0,Y 394.576,Z 580.237,A -85,B 0,C 180,E1 -24835.349,E2 -24835.349} C_VEL
LIN {X 0,Y 393.231,Z 576.445,A -85,B 0,C 180,E1 -24840.874,E2 -24840.874} C_VEL
LIN {X 0,Y 393.327,Z 577.972,A -85,B 0,C 180,E1 -24843.003,E2 -24843.003} C_VEL
LIN {X 0,Y 393.472,Z 579.728,A -85,B 0,C 180,E1 -24844.107,E2 -24844.107} C_VEL
LIN {X 0,Y 394.13,Z 589.269,A -85,B 0,C 180,E1 -24847.248,E2 -24847.248} C_VEL
LIN {X 0,Y 394.497,Z 590.432,A -85,B 0,C 180,E1 -24847.876,E2 -24847.876} C_VEL
LIN {X 0,Y 395.894,Z 593.101,A -85,B 0,C 180,E1 -24849.669,E2 -24849.669} C_VEL
LIN {X 0,Y 398.364,Z 598.093,A -85,B 0,C 180,E1 -24852.172,E2 -24852.172} C_VEL
LIN {X 0,Y 400.05,Z 601.908,A -85,B 0,C 180,E1 -24853.623,E2 -24853.623} C_VEL
LIN {X 0,Y 384.214,Z 755.061,A -85,B 0,C 180,E1 -24855.873,E2 -24855.873} C_VEL
LIN {X 0,Y 379.735,Z 781.548,A -85,B 0,C 180,E1 -24856.348,E2 -24856.348} C_VEL
LIN {X 0,Y 374.706,Z 803.088,A -85,B 0,C 180,E1 -24856.823,E2 -24856.823} C_VEL
LIN {X 0,Y 367.504,Z 827.537,A -85,B 0,C 180,E1 -24857.517,E2 -24857.517} C_VEL
LIN {X 0,Y 359.857,Z 848.846,A -85,B 0,C 180,E1 -24858.299,E2 -24858.299} C_VEL
LIN {X 0,Y 350.274,Z 871.762,A -85,B 0,C 180,E1 -24859.362,E2 -24859.362} C_VEL
LIN {X 0,Y 340.585,Z 891.671,A -85,B 0,C 180,E1 -24860.525,E2 -24860.525} C_VEL
LIN {X 0,Y 329.416,Z 912.179,A -85,B 0,C 180,E1 -24861.983,E2 -24861.983} C_VEL
LIN {X 0,Y 317.283,Z 931.705,A -85,B 0,C 180,E1 -24863.725,E2 -24863.725} C_VEL
LIN {X 0,Y 305.781,Z 948.621,A -85,B 0,C 180,E1 -24865.571,E2 -24865.571} C_VEL
LIN {X 0,Y 292.224,Z 966.7,A -85,B 0,C 180,E1 -24868.019,E2 -24868.019} C_VEL
LIN {X 0,Y 279.875,Z 981.832,A -85,B 0,C 180,E1 -24870.571,E2 -24870.571} C_VEL
LIN {X 0,Y 265.479,Z 998.208,A -85,B 0,C 180,E1 -24874.045,E2 -24874.045} C_VEL
LIN {X 0,Y 253.374,Z 1011.049,A -85,B 0,C 180,E1 -24877.514,E2 -24877.514} C_VEL
LIN {X 0,Y 240.617,Z 1024.011,A -85,B 0,C 180,E1 -24881.941,E2 -24881.941} C_VEL
LIN {X 0,Y 229.819,Z 1034.529,A -85,B 0,C 180,E1 -24886.601,E2 -24886.601} C_VEL
LIN {X 0,Y 219.857,Z 1044.319,A -85,B 0,C 180,E1 -24892.123,E2 -24892.123} C_VEL
LIN {X 0,Y 211.714,Z 1052.364,A -85,B 0,C 180,E1 -24898.224,E2 -24898.224} C_VEL
LIN {X 0,Y 205.808,Z 1058.873,A -85,B 0,C 180,E1 -24904.689,E2 -24904.689} C_VEL
LIN {X 0,Y 202.037,Z 1063.683,A -85,B 0,C 180,E1 -24911.534,E2 -24911.534} C_VEL
LIN {X 0,Y 200.463,Z 1066.504,A -85,B 0,C 180,E1 -24917.322,E2 -24917.322} C_VEL
LIN {X 0,Y 199.982,Z 1068.373,A -85,B 0,C 180,E1 -24923.685,E2 -24923.685} C_VEL
LIN {X 0,Y 200.023,Z 1068.819,A -85,B 0,C 180,E1 -24929.141,E2 -24929.141} C_VEL
LIN {X 0,Y 199.991,Z 1068.276,A -85,B 0,C 180,E1 -24934.301,E2 -24934.301} C_VEL
LIN {X 0,Y 200.137,Z 1066.573,A -85,B 0,C 180,E1 -24940.071,E2 -24940.071} C_VEL
LIN {X 0,Y 201.054,Z 1063.923,A -85,B 0,C 180,E1 -24945.578,E2 -24945.578} C_VEL
LIN {X 0,Y 203.56,Z 1059.605,A -85,B 0,C 180,E1 -24951.92,E2 -24951.92} C_VEL
LIN {X 0,Y 208.377,Z 1053.128,A -85,B 0,C 180,E1 -24958.675,E2 -24958.675} C_VEL
LIN {X 0,Y 214.622,Z 1045.879,A -85,B 0,C 180,E1 -24964.45,E2 -24964.45} C_VEL
LIN {X 0,Y 224.021,Z 1035.644,A -85,B 0,C 180,E1 -24970.666,E2 -24970.666} C_VEL
LIN {X 0,Y 233.324,Z 1025.711,A -85,B 0,C 180,E1 -24975.347,E2 -24975.347} C_VEL
LIN {X 0,Y 245.68,Z 1012.315,A -85,B 0,C 180,E1 -24980.285,E2 -24980.285} C_VEL
LIN {X 0,Y 256.46,Z 1000.167,A -85,B 0,C 180,E1 -24983.809,E2 -24983.809} C_VEL
LIN {X 0,Y 269.465,Z 984.83,A -85,B 0,C 180,E1 -24987.386,E2 -24987.386} C_VEL
LIN {X 0,Y 281.973,Z 968.866,A -85,B 0,C 180,E1 -24990.317,E2 -24990.317} C_VEL
LIN {X 0,Y 294.793,Z 951.371,A -85,B 0,C 180,E1 -24992.918,E2 -24992.918} C_VEL
LIN {X 0,Y 306.993,Z 932.839,A -85,B 0,C 180,E1 -24995.106,E2 -24995.106} C_VEL
LIN {X 0,Y 318.827,Z 913.227,A -85,B 0,C 180,E1 -24996.993,E2 -24996.993} C_VEL
LIN {X 0,Y 329.766,Z 892.633,A -85,B 0,C 180,E1 -24998.569,E2 -24998.569} C_VEL
LIN {X 0,Y 339.294,Z 872.562,A -85,B 0,C 180,E1 -24999.831,E2 -24999.831} C_VEL
LIN {X 0,Y 348.535,Z 850.03,A -85,B 0,C 180,E1 -25000.958,E2 -25000.958} C_VEL
LIN {X 0,Y 355.376,Z 830.704,A -85,B 0,C 180,E1 -25001.73,E2 -25001.73} C_VEL
LIN {X 0,Y 362.468,Z 807.01,A -85,B 0,C 180,E1 -25002.488,E2 -25002.488} C_VEL
LIN {X 0,Y 367.851,Z 783.923,A -85,B 0,C 180,E1 -25003.048,E2 -25003.048} C_VEL
LIN {X 0,Y 372.199,Z 759.171,A -85,B 0,C 180,E1 -25003.531,E2 -25003.531} C_VEL
LIN {X 0,Y 377.685,Z 706.461,A -85,B 0,C 180,E1 -25004.353,E2 -25004.353} C_VEL
LIN {X 0,Y 388.874,Z 592.849,A -85,B 0,C 180,E1 -25006.089,E2 -25006.089} C_VEL
LIN {X 0,Y 385.178,Z 585.215,A -85,B 0,C 180,E1 -25008.925,E2 -25008.925} C_VEL
LIN {X 0,Y 382.747,Z 580.59,A -85,B 0,C 180,E1 -25011.209,E2 -25011.209} C_VEL
LIN {X 0,Y 381.276,Z 577.69,A -85,B 0,C 180,E1 -25012.92,E2 -25012.92} C_VEL
LIN {X 0,Y 379.622,Z 574.257,A -85,B 0,C 180,E1 -25015.468,E2 -25015.468} C_VEL
LIN {X 0,Y 378.213,Z 570.273,A -85,B 0,C 180,E1 -25021.363,E2 -25021.363} C_VEL
LIN {X 0,Y 379.97,Z 574.909,A -85,B 0,C 180,E1 -25027.561,E2 -25027.561} C_VEL
LIN {X 0,Y 382.225,Z 579.469,A -85,B 0,C 180,E1 -25030.628,E2 -25030.628} C_VEL
LIN {X 0,Y 384.766,Z 584.495,A -85,B 0,C 180,E1 -25033.143,E2 -25033.143} C_VEL
LIN {X 0,Y 388.192,Z 591.377,A -85,B 0,C 180,E1 -25035.845,E2 -25035.845} C_VEL
LIN {X 0,Y 388.843,Z 592.94,A -85,B 0,C 180,E1 -25036.317,E2 -25036.317} C_VEL
LIN {X 0,Y 373.131,Z 749.354,A -85,B 0,C 180,E1 -25038.68,E2 -25038.68} C_VEL
LIN {X 0,Y 368.838,Z 775.592,A -85,B 0,C 180,E1 -25039.193,E2 -25039.193} C_VEL
LIN {X 0,Y 364.12,Z 796.672,A -85,B 0,C 180,E1 -25039.734,E2 -25039.734} C_VEL
LIN {X 0,Y 357.192,Z 821.284,A -85,B 0,C 180,E1 -25040.55,E2 -25040.55} C_VEL
LIN {X 0,Y 349.774,Z 842.796,A -85,B 0,C 180,E1 -25041.464,E2 -25041.464} C_VEL
LIN {X 0,Y 340.742,Z 865.252,A -85,B 0,C 180,E1 -25042.649,E2 -25042.649} C_VEL
LIN {X 0,Y 331.462,Z 884.983,A -85,B 0,C 180,E1 -25043.932,E2 -25043.932} C_VEL
LIN {X 0,Y 321.189,Z 904.555,A -85,B 0,C 180,E1 -25045.472,E2 -25045.472} C_VEL
LIN {X 0,Y 309.619,Z 923.998,A -85,B 0,C 180,E1 -25047.366,E2 -25047.366} C_VEL
LIN {X 0,Y 298.756,Z 940.592,A -85,B 0,C 180,E1 -25049.325,E2 -25049.325} C_VEL
LIN {X 0,Y 285.424,Z 959.111,A -85,B 0,C 180,E1 -25052.03,E2 -25052.03} C_VEL
LIN {X 0,Y 274.417,Z 973.146,A -85,B 0,C 180,E1 -25054.566,E2 -25054.566} C_VEL
LIN {X 0,Y 261.441,Z 988.661,A -85,B 0,C 180,E1 -25058.015,E2 -25058.015} C_VEL
LIN {X 0,Y 249.428,Z 1001.97,A -85,B 0,C 180,E1 -25061.787,E2 -25061.787} C_VEL
LIN {X 0,Y 238.014,Z 1014.207,A -85,B 0,C 180,E1 -25066.119,E2 -25066.119} C_VEL
LIN {X 0,Y 227.439,Z 1025.012,A -85,B 0,C 180,E1 -25071.092,E2 -25071.092} C_VEL
LIN {X 0,Y 218.628,Z 1034.114,A -85,B 0,C 180,E1 -25076.4,E2 -25076.4} C_VEL
LIN {X 0,Y 210.957,Z 1042.177,A -85,B 0,C 180,E1 -25082.629,E2 -25082.629} C_VEL
LIN {X 0,Y 205.838,Z 1048.089,A -85,B 0,C 180,E1 -25088.634,E2 -25088.634} C_VEL
LIN {X 0,Y 202.099,Z 1053.164,A -85,B 0,C 180,E1 -25095.864,E2 -25095.864} C_VEL
LIN {X 0,Y 200.612,Z 1055.901,A -85,B 0,C 180,E1 -25101.689,E2 -25101.689} C_VEL
LIN {X 0,Y 200.103,Z 1057.542,A -85,B 0,C 180,E1 -25107.422,E2 -25107.422} C_VEL
LIN {X 0,Y 200.027,Z 1058.167,A -85,B 0,C 180,E1 -25113.152,E2 -25113.152} C_VEL
LIN {X 0,Y 200.279,Z 1057.583,A -85,B 0,C 180,E1 -25119.193,E2 -25119.193} C_VEL
LIN {X 0,Y 201.185,Z 1055.965,A -85,B 0,C 180,E1 -25124.978,E2 -25124.978} C_VEL
LIN {X 0,Y 203.399,Z 1053.134,A -85,B 0,C 180,E1 -25131.03,E2 -25131.03} C_VEL
LIN {X 0,Y 208.332,Z 1047.87,A -85,B 0,C 180,E1 -25138.369,E2 -25138.369} C_VEL
LIN {X 0,Y 214.24,Z 1042.154,A -85,B 0,C 180,E1 -25144.06,E2 -25144.06} C_VEL
LIN {X 0,Y 223.512,Z 1033.565,A -85,B 0,C 180,E1 -25150.441,E2 -25150.441} C_VEL
LIN {X 0,Y 233.081,Z 1024.672,A -85,B 0,C 180,E1 -25155.408,E2 -25155.408} C_VEL
LIN {X 0,Y 245.266,Z 1013.131,A -85,B 0,C 180,E1 -25160.4,E2 -25160.4} C_VEL
LIN {X 0,Y 256.9,Z 1001.514,A -85,B 0,C 180,E1 -25164.28,E2 -25164.28} C_VEL
LIN {X 0,Y 270.107,Z 987.682,A -85,B 0,C 180,E1 -25167.964,E2 -25167.964} C_VEL
LIN {X 0,Y 283.27,Z 972.632,A -85,B 0,C 180,E1 -25171.092,E2 -25171.092} C_VEL
LIN {X 0,Y 296.816,Z 956.045,A -85,B 0,C 180,E1 -25173.866,E2 -25173.866} C_VEL
LIN {X 0,Y 309.747,Z 938.391,A -85,B 0,C 180,E1 -25176.202,E2 -25176.202} C_VEL
LIN {X 0,Y 322.446,Z 919.477,A -85,B 0,C 180,E1 -25178.237,E2 -25178.237} C_VEL
LIN {X 0,Y 334.208,Z 899.531,A -85,B 0,C 180,E1 -25179.956,E2 -25179.956} C_VEL
LIN {X 0,Y 344.589,Z 879.973,A -85,B 0,C 180,E1 -25181.334,E2 -25181.334} C_VEL
LIN {X 0,Y 354.703,Z 857.899,A -85,B 0,C 180,E1 -25182.595,E2 -25182.595} C_VEL
LIN {X 0,Y 362.288,Z 838.902,A -85,B 0,C 180,E1 -25183.484,E2 -25183.484} C_VEL
LIN {X 0,Y 370.59,Z 814.284,A -85,B 0,C 180,E1 -25184.413,E2 -25184.413} C_VEL
LIN {X 0,Y 376.483,Z 792.686,A -85,B 0,C 180,E1 -25185.051,E2 -25185.051} C_VEL
LIN {X 0,Y 381.88,Z 767.46,A -85,B 0,C 180,E1 -25185.619,E2 -25185.619} C_VEL
LIN {X 0,Y 385.279,Z 744.593,A -85,B 0,C 180,E1 -25186.009,E2 -25186.009} C_VEL
LIN {X 0,Y 399.969,Z 601.459,A -85,B 0,C 180,E1 -25188.131,E2 -25188.131} C_VEL
LIN {X 0,Y 396.863,Z 595.024,A -85,B 0,C 180,E1 -25190.94,E2 -25190.94} C_VEL
LIN {X 0,Y 395.065,Z 591.422,A -85,B 0,C 180,E1 -25193.022,E2 -25193.022} C_VEL
LIN {X 0,Y 393.517,Z 588.118,A -85,B 0,C 180,E1 -25195.482,E2 -25195.482} C_VEL
LIN {X 0,Y 392.243,Z 584.508,A -85,B 0,C 180,E1 -25201.022,E2 -25201.022} C_VEL
LIN {X 0,Y 393.803,Z 588.669,A -85,B 0,C 180,E1 -25206.707,E2 -25206.707} C_VEL
LIN {X 0,Y 394.497,Z 590.432,A -85,B 0,C 180,E1 -25207.876,E2 -25207.876} C_VEL
LIN {X 0,Y 394.865,Z 592.475,A -85,B 0,C 180,E1 -25208.571,E2 -25208.571} C_VEL
LIN {X 0,Y 395.442,Z 601.545,A -85,B 0,C 180,E1 -25210.208,E2 -25210.208} C_VEL
LIN {X 0,Y 395.919,Z 603.34,A -85,B 0,C 180,E1 -25210.803,E2 -25210.803} C_VEL
LIN {X 0,Y 397.764,Z 607.479,A -85,B 0,C 180,E1 -25212.577,E2 -25212.577} C_VEL
LIN {X 0,Y 382.227,Z 754.858,A -85,B 0,C 180,E1 -25214.71,E2 -25214.71} C_VEL
LIN {X 0,Y 377.68,Z 781.364,A -85,B 0,C 180,E1 -25215.173,E2 -25215.173} C_VEL
LIN {X 0,Y 372.538,Z 803.082,A -85,B 0,C 180,E1 -25215.637,E2 -25215.637} C_VEL
LIN {X 0,Y 365.168,Z 827.678,A -85,B 0,C 180,E1 -25216.316,E2 -25216.316} C_VEL
LIN {X 0,Y 357.68,Z 848.26,A -85,B 0,C 180,E1 -25217.048,E2 -25217.048} C_VEL
LIN {X 0,Y 348.118,Z 870.897,A -85,B 0,C 180,E1 -25218.062,E2 -25218.062} C_VEL
LIN {X 0,Y 338.26,Z 890.87,A -85,B 0,C 180,E1 -25219.19,E2 -25219.19} C_VEL
LIN {X 0,Y 327.717,Z 909.962,A -85,B 0,C 180,E1 -25220.499,E2 -25220.499} C_VEL
LIN {X 0,Y 314.908,Z 930.438,A -85,B 0,C 180,E1 -25222.246,E2 -25222.246} C_VEL
LIN {X 0,Y 303.245,Z 947.288,A -85,B 0,C 180,E1 -25224.027,E2 -25224.027} C_VEL
LIN {X 0,Y 288.462,Z 966.61,A -85,B 0,C 180,E1 -25226.581,E2 -25226.581} C_VEL
LIN {X 0,Y 275.782,Z 981.731,A -85,B 0,C 180,E1 -25229.099,E2 -25229.099} C_VEL
LIN {X 0,Y 260.951,Z 998.085,A -85,B 0,C 180,E1 -25232.544,E2 -25232.544} C_VEL
LIN {X 0,Y 248.428,Z 1010.917,A -85,B 0,C 180,E1 -25236.002,E2 -25236.002} C_VEL
LIN {X 0,Y 235.162,Z 1023.861,A -85,B 0,C 180,E1 -25240.439,E2 -25240.439} C_VEL
LIN {X 0,Y 223.908,Z 1034.335,A -85,B 0,C 180,E1 -25245.124,E2 -25245.124} C_VEL
LIN {X 0,Y 213.377,Z 1044.148,A -85,B 0,C 180,E1 -25250.757,E2 -25250.757} C_VEL
LIN {X 0,Y 204.895,Z 1052.03,A -85,B 0,C 180,E1 -25256.869,E2 -25256.869} C_VEL
LIN {X 0,Y 198.394,Z 1058.688,A -85,B 0,C 180,E1 -25263.672,E2 -25263.672} C_VEL
LIN {X 0,Y 194.289,Z 1063.487,A -85,B 0,C 180,E1 -25270.769,E2 -25270.769} C_VEL
LIN {X 0,Y 192.492,Z 1066.42,A -85,B 0,C 180,E1 -25277.093,E2 -25277.093} C_VEL
LIN {X 0,Y 191.983,Z 1068.226,A -85,B 0,C 180,E1 -25283.721,E2 -25283.721} C_VEL
LIN {X 0,Y 192.028,Z 1068.581,A -85,B 0,C 180,E1 -25289.403,E2 -25289.403} C_VEL
LIN {X 0,Y 191.992,Z 1067.983,A -85,B 0,C 180,E1 -25294.78,E2 -25294.78} C_VEL
LIN {X 0,Y 192.171,Z 1066.342,A -85,B 0,C 180,E1 -25300.493,E2 -25300.493} C_VEL
LIN {X 0,Y 193.206,Z 1063.684,A -85,B 0,C 180,E1 -25306.228,E2 -25306.228} C_VEL
LIN {X 0,Y 196.132,Z 1059.144,A -85,B 0,C 180,E1 -25313.113,E2 -25313.113} C_VEL
LIN {X 0,Y 201.435,Z 1052.554,A -85,B 0,C 180,E1 -25320.089,E2 -25320.089} C_VEL
LIN {X 0,Y 208.411,Z 1045.038,A -85,B 0,C 180,E1 -25326.165,E2 -25326.165} C_VEL
LIN {X 0,Y 217.789,Z 1035.358,A -85,B 0,C 180,E1 -25332.09,E2 -25332.09} C_VEL
LIN {X 0,Y 227.563,Z 1025.418,A -85,B 0,C 180,E1 -25336.835,E2 -25336.835} C_VEL
LIN {X 0,Y 240.456,Z 1012.008,A -85,B 0,C 180,E1 -25341.806,E2 -25341.806} C_VEL
LIN {X 0,Y 251.991,Z 999.478,A -85,B 0,C 180,E1 -25345.429,E2 -25345.429} C_VEL
LIN {X 0,Y 265.797,Z 983.634,A -85,B 0,C 180,E1 -25349.06,E2 -25349.06} C_VEL
LIN {X 0,Y 277.981,Z 968.517,A -85,B 0,C 180,E1 -25351.794,E2 -25351.794} C_VEL
LIN {X 0,Y 291.141,Z 950.998,A -85,B 0,C 180,E1 -25354.359,E2 -25354.359} C_VEL
LIN {X 0,Y 303.234,Z 933.066,A -85,B 0,C 180,E1 -25356.446,E2 -25356.446} C_VEL
LIN {X 0,Y 314.492,Z 914.848,A -85,B 0,C 180,E1 -25358.184,E2 -25358.184} C_VEL
LIN {X 0,Y 326.04,Z 893.828,A -85,B 0,C 180,E1 -25359.79,E2 -25359.79} C_VEL
LIN {X 0,Y 335.282,Z 874.861,A -85,B 0,C 180,E1 -25360.973,E2 -25360.973} C_VEL
LIN {X 0,Y 345.114,Z 851.78,A -85,B 0,C 180,E1 -25362.129,E2 -25362.129} C_VEL
LIN {X 0,Y 352.486,Z 831.425,A -85,B 0,C 180,E1 -25362.932,E2 -25362.932} C_VEL
LIN {X 0,Y 359.498,Z 808.699,A -85,B 0,C 180,E1 -25363.651,E2 -25363.651} C_VEL
LIN {X 0,Y 365.249,Z 784.701,A -85,B 0,C 180,E1 -25364.225,E2 -25364.225} C_VEL
LIN {X 0,Y 369.558,Z 761.001,A -85,B 0,C 180,E1 -25364.682,E2 -25364.682} C_VEL
LIN {X 0,Y 373.795,Z 722.938,A -85,B 0,C 180,E1 -25365.277,E2 -25365.277} C_VEL
LIN {X 0,Y 386.335,Z 598.311,A -85,B 0,C 180,E1 -25367.139,E2 -25367.139} C_VEL
LIN {X 0,Y 383.013,Z 591.33,A -85,B 0,C 180,E1 -25369.927,E2 -25369.927} C_VEL
LIN {X 0,Y 380.415,Z 585.945,A -85,B 0,C 180,E1 -25372.752,E2 -25372.752} C_VEL
LIN {X 0,Y 378.474,Z 582.039,A -85,B 0,C 180,E1 -25375.758,E2 -25375.758} C_VEL
LIN {X 0,Y 377.231,Z 578.267,A -85,B 0,C 180,E1 -25381.367,E2 -25381.367} C_VEL
LIN {X 0,Y 378.855,Z 582.72,A -85,B 0,C 180,E1 -25387.354,E2 -25387.354} C_VEL
LIN {X 0,Y 380.974,Z 587.166,A -85,B 0,C 180,E1 -25390.357,E2 -25390.357} C_VEL
LIN {X 0,Y 383.435,Z 592.202,A -85,B 0,C 180,E1 -25392.883,E2 -25392.883} C_VEL
LIN {X 0,Y 386.293,Z 598.234,A -85,B 0,C 180,E1 -25395.247,E2 -25395.247} C_VEL
LIN {X 0,Y 370.781,Z 749.609,A -85,B 0,C 180,E1 -25397.502,E2 -25397.502} C_VEL
LIN {X 0,Y 366.405,Z 775.895,A -85,B 0,C 180,E1 -25398.005,E2 -25398.005} C_VEL
LIN {X 0,Y 361.614,Z 796.958,A -85,B 0,C 180,E1 -25398.532,E2 -25398.532} C_VEL
LIN {X 0,Y 354.469,Z 821.873,A -85,B 0,C 180,E1 -25399.342,E2 -25399.342} C_VEL
LIN {X 0,Y 347.304,Z 842.342,A -85,B 0,C 180,E1 -25400.19,E2 -25400.19} C_VEL
LIN {X 0,Y 338.154,Z 864.84,A -85,B 0,C 180,E1 -25401.342,E2 -25401.342} C_VEL
LIN {X 0,Y 328.289,Z 885.437,A -85,B 0,C 180,E1 -25402.651,E2 -25402.651} C_VEL
LIN {X 0,Y 317.416,Z 905.713,A -85,B 0,C 180,E1 -25404.223,E2 -25404.223} C_VEL
LIN {X 0,Y 305.607,Z 924.995,A -85,B 0,C 180,E1 -25406.089,E2 -25406.089} C_VEL
LIN {X 0,Y 294.254,Z 941.888,A -85,B 0,C 180,E1 -25408.072,E2 -25408.072} C_VEL
LIN {X 0,Y 281.209,Z 959.465,A -85,B 0,C 180,E1 -25410.63,E2 -25410.63} C_VEL
LIN {X 0,Y 269.204,Z 974.323,A -85,B 0,C 180,E1 -25413.311,E2 -25413.311} C_VEL
LIN {X 0,Y 255.218,Z 990.363,A -85,B 0,C 180,E1 -25416.943,E2 -25416.943} C_VEL
LIN {X 0,Y 243.481,Z 1002.907,A -85,B 0,C 180,E1 -25420.56,E2 -25420.56} C_VEL
LIN {X 0,Y 230.949,Z 1015.708,A -85,B 0,C 180,E1 -25425.238,E2 -25425.238} C_VEL
LIN {X 0,Y 220.75,Z 1025.688,A -85,B 0,C 180,E1 -25429.97,E2 -25429.97} C_VEL
LIN {X 0,Y 211.127,Z 1035.168,A -85,B 0,C 180,E1 -25435.696,E2 -25435.696} C_VEL
LIN {X 0,Y 203.473,Z 1042.736,A -85,B 0,C 180,E1 -25441.852,E2 -25441.852} C_VEL
LIN {X 0,Y 197.87,Z 1048.88,A -85,B 0,C 180,E1 -25448.405,E2 -25448.405} C_VEL
LIN {X 0,Y 194.225,Z 1053.482,A -85,B 0,C 180,E1 -25455.432,E2 -25455.432} C_VEL
LIN {X 0,Y 192.665,Z 1056.132,A -85,B 0,C 180,E1 -25461.344,E2 -25461.344} C_VEL
LIN {X 0,Y 192.109,Z 1057.766,A -85,B 0,C 180,E1 -25467.315,E2 -25467.315} C_VEL
LIN {X 0,Y 192.031,Z 1058.383,A -85,B 0,C 180,E1 -25473.284,E2 -25473.284} C_VEL
LIN {X 0,Y 192.288,Z 1057.854,A -85,B 0,C 180,E1 -25479.277,E2 -25479.277} C_VEL
LIN {X 0,Y 193.332,Z 1056.165,A -85,B 0,C 180,E1 -25485.601,E2 -25485.601} C_VEL
LIN {X 0,Y 195.766,Z 1053.328,A -85,B 0,C 180,E1 -25491.892,E2 -25491.892} C_VEL
LIN {X 0,Y 201.105,Z 1048.051,A -85,B 0,C 180,E1 -25499.487,E2 -25499.487} C_VEL
LIN {X 0,Y 207.429,Z 1042.328,A -85,B 0,C 180,E1 -25505.341,E2 -25505.341} C_VEL
LIN {X 0,Y 217.266,Z 1033.724,A -85,B 0,C 180,E1 -25511.86,E2 -25511.86} C_VEL
LIN {X 0,Y 227.331,Z 1024.823,A -85,B 0,C 180,E1 -25516.898,E2 -25516.898} C_VEL
LIN {X 0,Y 240.184,Z 1013.15,A -85,B 0,C 180,E1 -25521.966,E2 -25521.966} C_VEL
LIN {X 0,Y 252.413,Z 1001.383,A -85,B 0,C 180,E1 -25525.885,E2 -25525.885} C_VEL
LIN {X 0,Y 265.872,Z 987.724,A -85,B 0,C 180,E1 -25529.489,E2 -25529.489} C_VEL
LIN {X 0,Y 279.379,Z 972.724,A -85,B 0,C 180,E1 -25532.572,E2 -25532.572} C_VEL
LIN {X 0,Y 293.373,Z 956.006,A -85,B 0,C 180,E1 -25535.322,E2 -25535.322} C_VEL
LIN {X 0,Y 306.579,Z 938.377,A -85,B 0,C 180,E1 -25537.611,E2 -25537.611} C_VEL
LIN {X 0,Y 319.51,Z 919.5,A -85,B 0,C 180,E1 -25539.598,E2 -25539.598} C_VEL
LIN {X 0,Y 331.503,Z 899.528,A -85,B 0,C 180,E1 -25541.28,E2 -25541.28} C_VEL
LIN {X 0,Y 342.502,Z 879.137,A -85,B 0,C 180,E1 -25542.676,E2 -25542.676} C_VEL
LIN {X 0,Y 352.348,Z 857.848,A -85,B 0,C 180,E1 -25543.853,E2 -25543.853} C_VEL
LIN {X 0,Y 360.134,Z 838.623,A -85,B 0,C 180,E1 -25544.725,E2 -25544.725} C_VEL
LIN {X 0,Y 368.502,Z 814.062,A -85,B 0,C 180,E1 -25545.622,E2 -25545.622} C_VEL
LIN {X 0,Y 374.417,Z 792.649,A -85,B 0,C 180,E1 -25546.237,E2 -25546.237} C_VEL
LIN {X 0,Y 379.943,Z 766.994,A -85,B 0,C 180,E1 -25546.796,E2 -25546.796} C_VEL
LIN {X 0,Y 383.326,Z 744.44,A -85,B 0,C 180,E1 -25547.17,E2 -25547.17} C_VEL
LIN {X 0,Y 397.689,Z 607.171,A -85,B 0,C 180,E1 -25549.167,E2 -25549.167} C_VEL
LIN {X 0,Y 395.192,Z 601.942,A -85,B 0,C 180,E1 -25551.635,E2 -25551.635} C_VEL
LIN {X 0,Y 393.858,Z 599.124,A -85,B 0,C 180,E1 -25553.294,E2 -25553.294} C_VEL
LIN {X 0,Y 392.459,Z 596,A -85,B 0,C 180,E1 -25555.616,E2 -25555.616} C_VEL
LIN {X 0,Y 391.263,Z 592.483,A -85,B 0,C 180,E1 -25561.025,E2 -25561.025} C_VEL
LIN {X 0,Y 392.699,Z 596.479,A -85,B 0,C 180,E1 -25566.506,E2 -25566.506} C_VEL
LIN {X 0,Y 394.717,Z 600.935,A -85,B 0,C 180,E1 -25569.477,E2 -25569.477} C_VEL
LIN {X 0,Y 395.919,Z 603.34,A -85,B 0,C 180,E1 -25570.803,E2 -25570.803} C_VEL
LIN {X 0,Y 396.183,Z 604.959,A -85,B 0,C 180,E1 -25571.178,E2 -25571.178} C_VEL
LIN {X 0,Y 396.148,Z 608.307,A -85,B 0,C 180,E1 -25571.476,E2 -25571.476} C_VEL
LIN {X 0,Y 395.721,Z 613.49,A -85,B 0,C 180,E1 -25571.645,E2 -25571.645} C_VEL
LIN {X 0,Y 394.184,Z 626.449,A -85,B 0,C 180,E1 -25571.708,E2 -25571.708} C_VEL
LIN {X 0,Y 380.379,Z 754.832,A -85,B 0,C 180,E1 -25573.537,E2 -25573.537} C_VEL
LIN {X 0,Y 375.788,Z 781.17,A -85,B 0,C 180,E1 -25573.986,E2 -25573.986} C_VEL
LIN {X 0,Y 370.573,Z 802.914,A -85,B 0,C 180,E1 -25574.435,E2 -25574.435} C_VEL
LIN {X 0,Y 362.861,Z 828.205,A -85,B 0,C 180,E1 -25575.113,E2 -25575.113} C_VEL
LIN {X 0,Y 355.143,Z 849.027,A -85,B 0,C 180,E1 -25575.835,E2 -25575.835} C_VEL
LIN {X 0,Y 344.823,Z 872.731,A -85,B 0,C 180,E1 -25576.882,E2 -25576.882} C_VEL
LIN {X 0,Y 334.825,Z 892.502,A -85,B 0,C 180,E1 -25577.985,E2 -25577.985} C_VEL
LIN {X 0,Y 322.843,Z 913.487,A -85,B 0,C 180,E1 -25579.425,E2 -25579.425} C_VEL
LIN {X 0,Y 310.673,Z 932.218,A -85,B 0,C 180,E1 -25581.036,E2 -25581.036} C_VEL
LIN {X 0,Y 297.194,Z 951.1,A -85,B 0,C 180,E1 -25583.049,E2 -25583.049} C_VEL
LIN {X 0,Y 283.332,Z 968.379,A -85,B 0,C 180,E1 -25585.387,E2 -25585.387} C_VEL
LIN {X 0,Y 268.909,Z 985.024,A -85,B 0,C 180,E1 -25588.208,E2 -25588.208} C_VEL
LIN {X 0,Y 254.505,Z 1000.079,A -85,B 0,C 180,E1 -25591.511,E2 -25591.511} C_VEL
LIN {X 0,Y 240.984,Z 1013.417,A -85,B 0,C 180,E1 -25595.222,E2 -25595.222} C_VEL
LIN {X 0,Y 227.523,Z 1025.793,A -85,B 0,C 180,E1 -25599.73,E2 -25599.73} C_VEL
LIN {X 0,Y 216.047,Z 1036.037,A -85,B 0,C 180,E1 -25604.543,E2 -25604.543} C_VEL
LIN {X 0,Y 204.88,Z 1045.773,A -85,B 0,C 180,E1 -25610.621,E2 -25610.621} C_VEL
LIN {X 0,Y 197.008,Z 1052.779,A -85,B 0,C 180,E1 -25616.412,E2 -25616.412} C_VEL
LIN {X 0,Y 189.904,Z 1059.588,A -85,B 0,C 180,E1 -25624.086,E2 -25624.086} C_VEL
LIN {X 0,Y 186.313,Z 1063.62,A -85,B 0,C 180,E1 -25630.565,E2 -25630.565} C_VEL
LIN {X 0,Y 184.372,Z 1066.692,A -85,B 0,C 180,E1 -25637.789,E2 -25637.789} C_VEL
LIN {X 0,Y 183.987,Z 1068.12,A -85,B 0,C 180,E1 -25644.699,E2 -25644.699} C_VEL
LIN {X 0,Y 184.042,Z 1068.32,A -85,B 0,C 180,E1 -25650,E2 -25650} C_VEL
LIN {X 0,Y 183.994,Z 1067.689,A -85,B 0,C 180,E1 -25655.301,E2 -25655.301} C_VEL
LIN {X 0,Y 184.213,Z 1066.11,A -85,B 0,C 180,E1 -25660.951,E2 -25660.951} C_VEL
LIN {X 0,Y 185.383,Z 1063.444,A -85,B 0,C 180,E1 -25666.933,E2 -25666.933} C_VEL
LIN {X 0,Y 188.729,Z 1058.733,A -85,B 0,C 180,E1 -25674.319,E2 -25674.319} C_VEL
LIN {X 0,Y 194.349,Z 1052.257,A -85,B 0,C 180,E1 -25681.346,E2 -25681.346} C_VEL
LIN {X 0,Y 201.777,Z 1044.768,A -85,B 0,C 180,E1 -25687.555,E2 -25687.555} C_VEL
LIN {X 0,Y 211.697,Z 1035.072,A -85,B 0,C 180,E1 -25693.597,E2 -25693.597} C_VEL
LIN {X 0,Y 221.962,Z 1025.124,A -85,B 0,C 180,E1 -25698.4,E2 -25698.4} C_VEL
LIN {X 0,Y 235.414,Z 1011.697,A -85,B 0,C 180,E1 -25703.394,E2 -25703.394} C_VEL
LIN {X 0,Y 247.035,Z 999.528,A -85,B 0,C 180,E1 -25706.913,E2 -25706.913} C_VEL
LIN {X 0,Y 260.925,Z 984.152,A -85,B 0,C 180,E1 -25710.445,E2 -25710.445} C_VEL
LIN {X 0,Y 273.425,Z 969.105,A -85,B 0,C 180,E1 -25713.162,E2 -25713.162} C_VEL
LIN {X 0,Y 286.498,Z 952.213,A -85,B 0,C 180,E1 -25715.63,E2 -25715.63} C_VEL
LIN {X 0,Y 299.686,Z 933.231,A -85,B 0,C 180,E1 -25717.825,E2 -25717.825} C_VEL
LIN {X 0,Y 311.129,Z 915.119,A -85,B 0,C 180,E1 -25719.522,E2 -25719.522} C_VEL
LIN {X 0,Y 323.314,Z 893.384,A -85,B 0,C 180,E1 -25721.146,E2 -25721.146} C_VEL
LIN {X 0,Y 332.718,Z 874.391,A -85,B 0,C 180,E1 -25722.298,E2 -25722.298} C_VEL
LIN {X 0,Y 343.146,Z 850.106,A -85,B 0,C 180,E1 -25723.47,E2 -25723.47} C_VEL
LIN {X 0,Y 350.637,Z 829.556,A -85,B 0,C 180,E1 -25724.244,E2 -25724.244} C_VEL
LIN {X 0,Y 358.045,Z 805.189,A -85,B 0,C 180,E1 -25724.965,E2 -25724.965} C_VEL
LIN {X 0,Y 363.333,Z 782.986,A -85,B 0,C 180,E1 -25725.469,E2 -25725.469} C_VEL
LIN {X 0,Y 367.777,Z 758.119,A -85,B 0,C 180,E1 -25725.929,E2 -25725.929} C_VEL
LIN {X 0,Y 373.825,Z 701.889,A -85,B 0,C 180,E1 -25726.776,E2 -25726.776} C_VEL
LIN {X 0,Y 383.88,Z 603.704,A -85,B 0,C 180,E1 -25728.24,E2 -25728.24} C_VEL
LIN {X 0,Y 380.828,Z 597.123,A -85,B 0,C 180,E1 -25731.088,E2 -25731.088} C_VEL
LIN {X 0,Y 378.954,Z 593.28,A -85,B 0,C 180,E1 -25733.333,E2 -25733.333} C_VEL
LIN {X 0,Y 377.415,Z 589.918,A -85,B 0,C 180,E1 -25735.898,E2 -25735.898} C_VEL
LIN {X 0,Y 376.262,Z 586.148,A -85,B 0,C 180,E1 -25741.218,E2 -25741.218} C_VEL
LIN {X 0,Y 377.784,Z 590.646,A -85,B 0,C 180,E1 -25747.222,E2 -25747.222} C_VEL
LIN {X 0,Y 379.731,Z 594.863,A -85,B 0,C 180,E1 -25750.085,E2 -25750.085} C_VEL
LIN {X 0,Y 382.439,Z 600.521,A -85,B 0,C 180,E1 -25752.917,E2 -25752.917} C_VEL
LIN {X 0,Y 383.853,Z 603.775,A -85,B 0,C 180,E1 -25754.166,E2 -25754.166} C_VEL
LIN {X 0,Y 368.589,Z 749.865,A -85,B 0,C 180,E1 -25756.309,E2 -25756.309} C_VEL
LIN {X 0,Y 364.159,Z 776.069,A -85,B 0,C 180,E1 -25756.799,E2 -25756.799} C_VEL
LIN {X 0,Y 359.246,Z 797.335,A -85,B 0,C 180,E1 -25757.317,E2 -25757.317} C_VEL
LIN {X 0,Y 351.905,Z 822.461,A -85,B 0,C 180,E1 -25758.115,E2 -25758.115} C_VEL
LIN {X 0,Y 344.628,Z 842.885,A -85,B 0,C 180,E1 -25758.943,E2 -25758.943} C_VEL
LIN {X 0,Y 335.322,Z 865.317,A -85,B 0,C 180,E1 -25760.067,E2 -25760.067} C_VEL
LIN {X 0,Y 325.283,Z 885.89,A -85,B 0,C 180,E1 -25761.347,E2 -25761.347} C_VEL
LIN {X 0,Y 314.2,Z 906.14,A -85,B 0,C 180,E1 -25762.885,E2 -25762.885} C_VEL
LIN {X 0,Y 302.146,Z 925.391,A -85,B 0,C 180,E1 -25764.715,E2 -25764.715} C_VEL
LIN {X 0,Y 290.027,Z 942.998,A -85,B 0,C 180,E1 -25766.757,E2 -25766.757} C_VEL
LIN {X 0,Y 276.426,Z 960.733,A -85,B 0,C 180,E1 -25769.338,E2 -25769.338} C_VEL
LIN {X 0,Y 264.126,Z 975.499,A -85,B 0,C 180,E1 -25772.007,E2 -25772.007} C_VEL
LIN {X 0,Y 249.749,Z 991.375,A -85,B 0,C 180,E1 -25775.637,E2 -25775.637} C_VEL
LIN {X 0,Y 238.266,Z 1003.221,A -85,B 0,C 180,E1 -25779.072,E2 -25779.072} C_VEL
LIN {X 0,Y 225.426,Z 1015.823,A -85,B 0,C 180,E1 -25783.698,E2 -25783.698} C_VEL
LIN {X 0,Y 214.568,Z 1025.975,A -85,B 0,C 180,E1 -25788.569,E2 -25788.569} C_VEL
LIN {X 0,Y 204.441,Z 1035.44,A -85,B 0,C 180,E1 -25794.408,E2 -25794.408} C_VEL
LIN {X 0,Y 196.331,Z 1042.999,A -85,B 0,C 180,E1 -25800.731,E2 -25800.731} C_VEL
LIN {X 0,Y 190.381,Z 1049.094,A -85,B 0,C 180,E1 -25807.456,E2 -25807.456} C_VEL
LIN {X 0,Y 186.436,Z 1053.7,A -85,B 0,C 180,E1 -25814.764,E2 -25814.764} C_VEL
LIN {X 0,Y 184.724,Z 1056.364,A -85,B 0,C 180,E1 -25820.969,E2 -25820.969} C_VEL
LIN {X 0,Y 184.116,Z 1057.99,A -85,B 0,C 180,E1 -25827.199,E2 -25827.199} C_VEL
LIN {X 0,Y 184.031,Z 1058.577,A -85,B 0,C 180,E1 -25833.115,E2 -25833.115} C_VEL
LIN {X 0,Y 184.297,Z 1058.124,A -85,B 0,C 180,E1 -25839.367,E2 -25839.367} C_VEL
LIN {X 0,Y 185.411,Z 1056.475,A -85,B 0,C 180,E1 -25845.964,E2 -25845.964} C_VEL
LIN {X 0,Y 187.847,Z 1053.833,A -85,B 0,C 180,E1 -25852.205,E2 -25852.205} C_VEL
LIN {X 0,Y 192.889,Z 1049.228,A -85,B 0,C 180,E1 -25859.502,E2 -25859.502} C_VEL
LIN {X 0,Y 200.005,Z 1043.098,A -85,B 0,C 180,E1 -25866.151,E2 -25866.151} C_VEL
LIN {X 0,Y 209.332,Z 1035.472,A -85,B 0,C 180,E1 -25872.338,E2 -25872.338} C_VEL
LIN {X 0,Y 220.668,Z 1025.882,A -85,B 0,C 180,E1 -25877.998,E2 -25877.998} C_VEL
LIN {X 0,Y 233.222,Z 1015.086,A -85,B 0,C 180,E1 -25882.886,E2 -25882.886} C_VEL
LIN {X 0,Y 246.535,Z 1002.768,A -85,B 0,C 180,E1 -25887.092,E2 -25887.092} C_VEL
LIN {X 0,Y 259.579,Z 990.037,A -85,B 0,C 180,E1 -25890.522,E2 -25890.522} C_VEL
LIN {X 0,Y 274.176,Z 974.5,A -85,B 0,C 180,E1 -25893.784,E2 -25893.784} C_VEL
LIN {X 0,Y 286.421,Z 960.373,A -85,B 0,C 180,E1 -25896.154,E2 -25896.154} C_VEL
LIN {X 0,Y 301.525,Z 941.2,A -85,B 0,C 180,E1 -25898.721,E2 -25898.721} C_VEL
LIN {X 0,Y 313.493,Z 924.303,A -85,B 0,C 180,E1 -25900.525,E2 -25900.525} C_VEL
LIN {X 0,Y 326.855,Z 903.201,A -85,B 0,C 180,E1 -25902.349,E2 -25902.349} C_VEL
LIN {X 0,Y 337.283,Z 884.528,A -85,B 0,C 180,E1 -25903.642,E2 -25903.642} C_VEL
LIN {X 0,Y 348.01,Z 862.771,A -85,B 0,C 180,E1 -25904.88,E2 -25904.88} C_VEL
LIN {X 0,Y 356.801,Z 841.79,A -85,B 0,C 180,E1 -25905.841,E2 -25905.841} C_VEL
LIN {X 0,Y 364.795,Z 819.642,A -85,B 0,C 180,E1 -25906.666,E2 -25906.666} C_VEL
LIN {X 0,Y 371.693,Z 795.793,A -85,B 0,C 180,E1 -25907.355,E2 -25907.355} C_VEL
LIN {X 0,Y 376.98,Z 772.958,A -85,B 0,C 180,E1 -25907.863,E2 -25907.863} C_VEL
LIN {X 0,Y 381.079,Z 747.849,A -85,B 0,C 180,E1 -25908.289,E2 -25908.289} C_VEL
LIN {X 0,Y 395.525,Z 613.102,A -85,B 0,C 180,E1 -25910.208,E2 -25910.208} C_VEL
LIN {X 0,Y 393.149,Z 607.705,A -85,B 0,C 180,E1 -25912.914,E2 -25912.914} C_VEL
LIN {X 0,Y 391.328,Z 603.79,A -85,B 0,C 180,E1 -25915.897,E2 -25915.897} C_VEL
LIN {X 0,Y 390.283,Z 600.464,A -85,B 0,C 180,E1 -25921.028,E2 -25921.028} C_VEL
LIN {X 0,Y 391.634,Z 604.404,A -85,B 0,C 180,E1 -25926.376,E2 -25926.376} C_VEL
LIN {X 0,Y 393.488,Z 608.629,A -85,B 0,C 180,E1 -25929.212,E2 -25929.212} C_VEL
LIN {X 0,Y 395.592,Z 613.189,A -85,B 0,C 180,E1 -25931.518,E2 -25931.518} C_VEL
LIN {X 0,Y 394.184,Z 626.449,A -85,B 0,C 180,E1 -25931.708,E2 -25931.708} C_VEL
LIN {X 0,Y 393.172,Z 634.147,A -85,B 0,C 180,E1 -25931.67,E2 -25931.67} C_VEL
LIN {X 0,Y 389.82,Z 654.704,A -85,B 0,C 180,E1 -25931.054,E2 -25931.054} C_VEL
LIN {X 0,Y 388.977,Z 661.307,A -85,B 0,C 180,E1 -25931.038,E2 -25931.038} C_VEL
LIN {X 0,Y 378.64,Z 755.206,A -85,B 0,C 180,E1 -25932.359,E2 -25932.359} C_VEL
LIN {X 0,Y 374.022,Z 781.147,A -85,B 0,C 180,E1 -25932.79,E2 -25932.79} C_VEL
LIN {X 0,Y 368.738,Z 802.884,A -85,B 0,C 180,E1 -25933.224,E2 -25933.224} C_VEL
LIN {X 0,Y 360.827,Z 828.417,A -85,B 0,C 180,E1 -25933.885,E2 -25933.885} C_VEL
LIN {X 0,Y 352.851,Z 849.587,A -85,B 0,C 180,E1 -25934.597,E2 -25934.597} C_VEL
LIN {X 0,Y 342.123,Z 873.665,A -85,B 0,C 180,E1 -25935.635,E2 -25935.635} C_VEL
LIN {X 0,Y 332.417,Z 892.512,A -85,B 0,C 180,E1 -25936.659,E2 -25936.659} C_VEL
LIN {X 0,Y 320.236,Z 913.457,A -85,B 0,C 180,E1 -25938.056,E2 -25938.056} C_VEL
LIN {X 0,Y 308.266,Z 931.562,A -85,B 0,C 180,E1 -25939.564,E2 -25939.564} C_VEL
LIN {X 0,Y 295.322,Z 949.387,A -85,B 0,C 180,E1 -25941.396,E2 -25941.396} C_VEL
LIN {X 0,Y 280.673,Z 967.403,A -85,B 0,C 180,E1 -25943.738,E2 -25943.738} C_VEL
LIN {X 0,Y 267.373,Z 982.413,A -85,B 0,C 180,E1 -25946.186,E2 -25946.186} C_VEL
LIN {X 0,Y 251.736,Z 998.546,A -85,B 0,C 180,E1 -25949.557,E2 -25949.557} C_VEL
LIN {X 0,Y 239.086,Z 1010.653,A -85,B 0,C 180,E1 -25952.796,E2 -25952.796} C_VEL
LIN {X 0,Y 224.157,Z 1024.084,A -85,B 0,C 180,E1 -25957.439,E2 -25957.439} C_VEL
LIN {X 0,Y 211.935,Z 1034.486,A -85,B 0,C 180,E1 -25962.208,E2 -25962.208} C_VEL
LIN {X 0,Y 199.895,Z 1044.523,A -85,B 0,C 180,E1 -25968.296,E2 -25968.296} C_VEL
LIN {X 0,Y 190.89,Z 1051.982,A -85,B 0,C 180,E1 -25974.449,E2 -25974.449} C_VEL
LIN {X 0,Y 183.512,Z 1058.546,A -85,B 0,C 180,E1 -25981.704,E2 -25981.704} C_VEL
LIN {X 0,Y 178.898,Z 1063.093,A -85,B 0,C 180,E1 -25989.041,E2 -25989.041} C_VEL
LIN {X 0,Y 176.682,Z 1066.017,A -85,B 0,C 180,E1 -25995.916,E2 -25995.916} C_VEL
LIN {X 0,Y 175.988,Z 1067.831,A -85,B 0,C 180,E1 -26003.475,E2 -26003.475} C_VEL
LIN {X 0,Y 176.033,Z 1068.148,A -85,B 0,C 180,E1 -26009.349,E2 -26009.349} C_VEL
LIN {X 0,Y 175.995,Z 1067.606,A -85,B 0,C 180,E1 -26014.889,E2 -26014.889} C_VEL
LIN {X 0,Y 176.226,Z 1065.996,A -85,B 0,C 180,E1 -26021.123,E2 -26021.123} C_VEL
LIN {X 0,Y 177.583,Z 1063.204,A -85,B 0,C 180,E1 -26027.701,E2 -26027.701} C_VEL
LIN {X 0,Y 181.31,Z 1058.414,A -85,B 0,C 180,E1 -26035.477,E2 -26035.477} C_VEL
LIN {X 0,Y 187.293,Z 1052.029,A -85,B 0,C 180,E1 -26042.629,E2 -26042.629} C_VEL
LIN {X 0,Y 195.674,Z 1044.135,A -85,B 0,C 180,E1 -26049.319,E2 -26049.319} C_VEL
LIN {X 0,Y 206.266,Z 1034.318,A -85,B 0,C 180,E1 -26055.446,E2 -26055.446} C_VEL
LIN {X 0,Y 217.687,Z 1023.781,A -85,B 0,C 180,E1 -26060.503,E2 -26060.503} C_VEL
LIN {X 0,Y 231.209,Z 1010.74,A -85,B 0,C 180,E1 -26065.253,E2 -26065.253} C_VEL
LIN {X 0,Y 243.963,Z 997.829,A -85,B 0,C 180,E1 -26068.908,E2 -26068.908} C_VEL
LIN {X 0,Y 258.429,Z 982.098,A -85,B 0,C 180,E1 -26072.378,E2 -26072.378} C_VEL
LIN {X 0,Y 270.577,Z 967.817,A -85,B 0,C 180,E1 -26074.873,E2 -26074.873} C_VEL
LIN {X 0,Y 284.412,Z 950.248,A -85,B 0,C 180,E1 -26077.347,E2 -26077.347} C_VEL
LIN {X 0,Y 297.06,Z 932.287,A -85,B 0,C 180,E1 -26079.347,E2 -26079.347} C_VEL
LIN {X 0,Y 309.095,Z 913.555,A -85,B 0,C 180,E1 -26081.04,E2 -26081.04} C_VEL
LIN {X 0,Y 320.773,Z 892.939,A -85,B 0,C 180,E1 -26082.524,E2 -26082.524} C_VEL
LIN {X 0,Y 330.464,Z 873.657,A -85,B 0,C 180,E1 -26083.657,E2 -26083.657} C_VEL
LIN {X 0,Y 340.926,Z 849.574,A -85,B 0,C 180,E1 -26084.777,E2 -26084.777} C_VEL
LIN {X 0,Y 348.526,Z 828.98,A -85,B 0,C 180,E1 -26085.525,E2 -26085.525} C_VEL
LIN {X 0,Y 356.134,Z 804.105,A -85,B 0,C 180,E1 -26086.23,E2 -26086.23} C_VEL
LIN {X 0,Y 361.393,Z 782.19,A -85,B 0,C 180,E1 -26086.708,E2 -26086.708} C_VEL
LIN {X 0,Y 365.893,Z 756.944,A -85,B 0,C 180,E1 -26087.159,E2 -26087.159} C_VEL
LIN {X 0,Y 372.896,Z 692.428,A -85,B 0,C 180,E1 -26088.11,E2 -26088.11} C_VEL
LIN {X 0,Y 381.599,Z 609.491,A -85,B 0,C 180,E1 -26089.295,E2 -26089.295} C_VEL
LIN {X 0,Y 379.208,Z 604.17,A -85,B 0,C 180,E1 -26091.738,E2 -26091.738} C_VEL
LIN {X 0,Y 377.638,Z 600.79,A -85,B 0,C 180,E1 -26093.768,E2 -26093.768} C_VEL
LIN {X 0,Y 376.358,Z 597.797,A -85,B 0,C 180,E1 -26096.039,E2 -26096.039} C_VEL
LIN {X 0,Y 375.281,Z 594.141,A -85,B 0,C 180,E1 -26101.221,E2 -26101.221} C_VEL
LIN {X 0,Y 376.678,Z 598.457,A -85,B 0,C 180,E1 -26107.014,E2 -26107.014} C_VEL
LIN {X 0,Y 378.554,Z 602.702,A -85,B 0,C 180,E1 -26109.886,E2 -26109.886} C_VEL
LIN {X 0,Y 381.113,Z 608.247,A -85,B 0,C 180,E1 -26112.655,E2 -26112.655} C_VEL
LIN {X 0,Y 381.528,Z 609.547,A -85,B 0,C 180,E1 -26113.076,E2 -26113.076} C_VEL
LIN {X 0,Y 366.559,Z 750.12,A -85,B 0,C 180,E1 -26115.103,E2 -26115.103} C_VEL
LIN {X 0,Y 362.076,Z 776.243,A -85,B 0,C 180,E1 -26115.579,E2 -26115.579} C_VEL
LIN {X 0,Y 357.091,Z 797.517,A -85,B 0,C 180,E1 -26116.081,E2 -26116.081} C_VEL
LIN {X 0,Y 349.506,Z 823.05,A -85,B 0,C 180,E1 -26116.871,E2 -26116.871} C_VEL
LIN {X 0,Y 342.117,Z 843.429,A -85,B 0,C 180,E1 -26117.677,E2 -26117.677} C_VEL
LIN {X 0,Y 332.658,Z 865.794,A -85,B 0,C 180,E1 -26118.771,E2 -26118.771} C_VEL
LIN {X 0,Y 322.871,Z 885.538,A -85,B 0,C 180,E1 -26119.965,E2 -26119.965} C_VEL
LIN {X 0,Y 311.943,Z 905.196,A -85,B 0,C 180,E1 -26121.409,E2 -26121.409} C_VEL
LIN {X 0,Y 299.268,Z 925.185,A -85,B 0,C 180,E1 -26123.248,E2 -26123.248} C_VEL
LIN {X 0,Y 287.263,Z 942.283,A -85,B 0,C 180,E1 -26125.177,E2 -26125.177} C_VEL
LIN {X 0,Y 273.305,Z 960.174,A -85,B 0,C 180,E1 -26127.704,E2 -26127.704} C_VEL
LIN {X 0,Y 260.637,Z 975.009,A -85,B 0,C 180,E1 -26130.325,E2 -26130.325} C_VEL
LIN {X 0,Y 245.784,Z 991.007,A -85,B 0,C 180,E1 -26133.911,E2 -26133.911} C_VEL
LIN {X 0,Y 233.332,Z 1003.421,A -85,B 0,C 180,E1 -26137.482,E2 -26137.482} C_VEL
LIN {X 0,Y 219.868,Z 1016.119,A -85,B 0,C 180,E1 -26142.16,E2 -26142.16} C_VEL
LIN {X 0,Y 208.522,Z 1026.262,A -85,B 0,C 180,E1 -26147.085,E2 -26147.085} C_VEL
LIN {X 0,Y 197.867,Z 1035.711,A -85,B 0,C 180,E1 -26153.033,E2 -26153.033} C_VEL
LIN {X 0,Y 189.27,Z 1043.262,A -85,B 0,C 180,E1 -26159.526,E2 -26159.526} C_VEL
LIN {X 0,Y 182.91,Z 1049.349,A -85,B 0,C 180,E1 -26166.481,E2 -26166.481} C_VEL
LIN {X 0,Y 178.653,Z 1053.939,A -85,B 0,C 180,E1 -26174.083,E2 -26174.083} C_VEL
LIN {X 0,Y 176.791,Z 1056.596,A -85,B 0,C 180,E1 -26180.56,E2 -26180.56} C_VEL
LIN {X 0,Y 176.123,Z 1058.214,A -85,B 0,C 180,E1 -26187.071,E2 -26187.071} C_VEL
LIN {X 0,Y 176.035,Z 1058.795,A -85,B 0,C 180,E1 -26193.256,E2 -26193.256} C_VEL
LIN {X 0,Y 176.331,Z 1058.329,A -85,B 0,C 180,E1 -26199.795,E2 -26199.795} C_VEL
LIN {X 0,Y 177.593,Z 1056.675,A -85,B 0,C 180,E1 -26206.687,E2 -26206.687} C_VEL
LIN {X 0,Y 180.275,Z 1054.027,A -85,B 0,C 180,E1 -26213.191,E2 -26213.191} C_VEL
LIN {X 0,Y 186.029,Z 1049.161,A -85,B 0,C 180,E1 -26221.064,E2 -26221.064} C_VEL
LIN {X 0,Y 193.375,Z 1043.272,A -85,B 0,C 180,E1 -26227.6,E2 -26227.6} C_VEL
LIN {X 0,Y 203.277,Z 1035.636,A -85,B 0,C 180,E1 -26233.912,E2 -26233.912} C_VEL
LIN {X 0,Y 214.645,Z 1026.486,A -85,B 0,C 180,E1 -26239.403,E2 -26239.403} C_VEL
LIN {X 0,Y 227.22,Z 1016.119,A -85,B 0,C 180,E1 -26244.178,E2 -26244.178} C_VEL
LIN {X 0,Y 241.451,Z 1003.523,A -85,B 0,C 180,E1 -26248.548,E2 -26248.548} C_VEL
LIN {X 0,Y 254.884,Z 990.848,A -85,B 0,C 180,E1 -26251.965,E2 -26251.965} C_VEL
LIN {X 0,Y 270.391,Z 974.862,A -85,B 0,C 180,E1 -26255.3,E2 -26255.3} C_VEL
LIN {X 0,Y 283.197,Z 960.454,A -85,B 0,C 180,E1 -26257.676,E2 -26257.676} C_VEL
LIN {X 0,Y 298.649,Z 941.253,A -85,B 0,C 180,E1 -26260.186,E2 -26260.186} C_VEL
LIN {X 0,Y 310.788,Z 924.449,A -85,B 0,C 180,E1 -26261.935,E2 -26261.935} C_VEL
LIN {X 0,Y 324.399,Z 903.332,A -85,B 0,C 180,E1 -26263.711,E2 -26263.711} C_VEL
LIN {X 0,Y 334.748,Z 885.127,A -85,B 0,C 180,E1 -26264.938,E2 -26264.938} C_VEL
LIN {X 0,Y 345.54,Z 863.698,A -85,B 0,C 180,E1 -26266.129,E2 -26266.129} C_VEL
LIN {X 0,Y 354.46,Z 842.805,A -85,B 0,C 180,E1 -26267.063,E2 -26267.063} C_VEL
LIN {X 0,Y 362.564,Z 820.768,A -85,B 0,C 180,E1 -26267.864,E2 -26267.864} C_VEL
LIN {X 0,Y 369.727,Z 796.587,A -85,B 0,C 180,E1 -26268.548,E2 -26268.548} C_VEL
LIN {X 0,Y 374.94,Z 774.526,A -85,B 0,C 180,E1 -26269.026,E2 -26269.026} C_VEL
LIN {X 0,Y 379.313,Z 748.676,A -85,B 0,C 180,E1 -26269.459,E2 -26269.459} C_VEL
LIN {X 0,Y 393.485,Z 619.026,A -85,B 0,C 180,E1 -26271.267,E2 -26271.267} C_VEL
LIN {X 0,Y 391.572,Z 614.717,A -85,B 0,C 180,E1 -26273.696,E2 -26273.696} C_VEL
LIN {X 0,Y 390.278,Z 611.67,A -85,B 0,C 180,E1 -26276.033,E2 -26276.033} C_VEL
LIN {X 0,Y 389.302,Z 608.455,A -85,B 0,C 180,E1 -26281.03,E2 -26281.03} C_VEL
LIN {X 0,Y 390.571,Z 612.326,A -85,B 0,C 180,E1 -26286.246,E2 -26286.246} C_VEL
LIN {X 0,Y 392.321,Z 616.461,A -85,B 0,C 180,E1 -26289.018,E2 -26289.018} C_VEL
LIN {X 0,Y 393.534,Z 619.198,A -85,B 0,C 180,E1 -26290.459,E2 -26290.459} C_VEL
LIN {X 0,Y 388.977,Z 661.307,A -85,B 0,C 180,E1 -26291.038,E2 -26291.038} C_VEL
LIN {X 0,Y 387.974,Z 669,A -85,B 0,C 180,E1 -26291.003,E2 -26291.003} C_VEL
LIN {X 0,Y 384.671,Z 689.552,A -85,B 0,C 180,E1 -26290.372,E2 -26290.372} C_VEL
LIN {X 0,Y 383.818,Z 696.159,A -85,B 0,C 180,E1 -26290.345,E2 -26290.345} C_VEL
LIN {X 0,Y 376.904,Z 756.796,A -85,B 0,C 180,E1 -26291.188,E2 -26291.188} C_VEL
LIN {X 0,Y 372.251,Z 781.89,A -85,B 0,C 180,E1 -26291.598,E2 -26291.598} C_VEL
LIN {X 0,Y 366.704,Z 804.231,A -85,B 0,C 180,E1 -26292.031,E2 -26292.031} C_VEL
LIN {X 0,Y 358.963,Z 828.627,A -85,B 0,C 180,E1 -26292.643,E2 -26292.643} C_VEL
LIN {X 0,Y 350.866,Z 849.8,A -85,B 0,C 180,E1 -26293.331,E2 -26293.331} C_VEL
LIN {X 0,Y 340.039,Z 873.702,A -85,B 0,C 180,E1 -26294.327,E2 -26294.327} C_VEL
LIN {X 0,Y 330.19,Z 892.523,A -85,B 0,C 180,E1 -26295.315,E2 -26295.315} C_VEL
LIN {X 0,Y 317.376,Z 914.095,A -85,B 0,C 180,E1 -26296.715,E2 -26296.715} C_VEL
LIN {X 0,Y 305.206,Z 932.124,A -85,B 0,C 180,E1 -26298.181,E2 -26298.181} C_VEL
LIN {X 0,Y 291.25,Z 950.871,A -85,B 0,C 180,E1 -26300.079,E2 -26300.079} C_VEL
LIN {X 0,Y 276.698,Z 968.201,A -85,B 0,C 180,E1 -26302.317,E2 -26302.317} C_VEL
LIN {X 0,Y 261.536,Z 984.812,A -85,B 0,C 180,E1 -26305.03,E2 -26305.03} C_VEL
LIN {X 0,Y 247.027,Z 999.13,A -85,B 0,C 180,E1 -26308.067,E2 -26308.067} C_VEL
LIN {X 0,Y 233.313,Z 1011.802,A -85,B 0,C 180,E1 -26311.478,E2 -26311.478} C_VEL
LIN {X 0,Y 217.945,Z 1024.975,A -85,B 0,C 180,E1 -26316.152,E2 -26316.152} C_VEL
LIN {X 0,Y 205.322,Z 1035.258,A -85,B 0,C 180,E1 -26320.989,E2 -26320.989} C_VEL
LIN {X 0,Y 192.83,Z 1045.07,A -85,B 0,C 180,E1 -26327.213,E2 -26327.213} C_VEL
LIN {X 0,Y 183.834,Z 1052.112,A -85,B 0,C 180,E1 -26333.252,E2 -26333.252} C_VEL
LIN {X 0,Y 175.756,Z 1058.78,A -85,B 0,C 180,E1 -26341.081,E2 -26341.081} C_VEL
LIN {X 0,Y 171.104,Z 1063.061,A -85,B 0,C 180,E1 -26348.398,E2 -26348.398} C_VEL
LIN {X 0,Y 168.662,Z 1066.053,A -85,B 0,C 180,E1 -26355.933,E2 -26355.933} C_VEL
LIN {X 0,Y 167.99,Z 1067.661,A -85,B 0,C 180,E1 -26363.722,E2 -26363.722} C_VEL
LIN {X 0,Y 168.04,Z 1067.91,A -85,B 0,C 180,E1 -26369.659,E2 -26369.659} C_VEL
LIN {X 0,Y 167.997,Z 1067.312,A -85,B 0,C 180,E1 -26375.464,E2 -26375.464} C_VEL
LIN {X 0,Y 168.321,Z 1065.647,A -85,B 0,C 180,E1 -26382,E2 -26382} C_VEL
LIN {X 0,Y 169.932,Z 1062.799,A -85,B 0,C 180,E1 -26388.882,E2 -26388.882} C_VEL
LIN {X 0,Y 174.136,Z 1057.897,A -85,B 0,C 180,E1 -26396.976,E2 -26396.976} C_VEL
LIN {X 0,Y 180.378,Z 1051.766,A -85,B 0,C 180,E1 -26404.047,E2 -26404.047} C_VEL
LIN {X 0,Y 189.469,Z 1043.746,A -85,B 0,C 180,E1 -26411.004,E2 -26411.004} C_VEL
LIN {X 0,Y 200.527,Z 1034.032,A -85,B 0,C 180,E1 -26417.137,E2 -26417.137} C_VEL
LIN {X 0,Y 212.499,Z 1023.486,A -85,B 0,C 180,E1 -26422.233,E2 -26422.233} C_VEL
LIN {X 0,Y 226.584,Z 1010.43,A -85,B 0,C 180,E1 -26426.976,E2 -26426.976} C_VEL
LIN {X 0,Y 239.836,Z 997.465,A -85,B 0,C 180,E1 -26430.614,E2 -26430.614} C_VEL
LIN {X 0,Y 254.701,Z 981.759,A -85,B 0,C 180,E1 -26434.026,E2 -26434.026} C_VEL
LIN {X 0,Y 267.18,Z 967.466,A -85,B 0,C 180,E1 -26436.474,E2 -26436.474} C_VEL
LIN {X 0,Y 281.346,Z 949.872,A -85,B 0,C 180,E1 -26438.893,E2 -26438.893} C_VEL
LIN {X 0,Y 294.267,Z 931.897,A -85,B 0,C 180,E1 -26440.841,E2 -26440.841} C_VEL
LIN {X 0,Y 306.661,Z 912.958,A -85,B 0,C 180,E1 -26442.5,E2 -26442.5} C_VEL
LIN {X 0,Y 318.42,Z 892.494,A -85,B 0,C 180,E1 -26443.923,E2 -26443.923} C_VEL
LIN {X 0,Y 328.138,Z 873.454,A -85,B 0,C 180,E1 -26445.005,E2 -26445.005} C_VEL
LIN {X 0,Y 338.437,Z 850.181,A -85,B 0,C 180,E1 -26446.056,E2 -26446.056} C_VEL
LIN {X 0,Y 346.137,Z 829.701,A -85,B 0,C 180,E1 -26446.779,E2 -26446.779} C_VEL
LIN {X 0,Y 353.642,Z 805.915,A -85,B 0,C 180,E1 -26447.441,E2 -26447.441} C_VEL
LIN {X 0,Y 359.282,Z 782.951,A -85,B 0,C 180,E1 -26447.93,E2 -26447.93} C_VEL
LIN {X 0,Y 363.861,Z 758.248,A -85,B 0,C 180,E1 -26448.363,E2 -26448.363} C_VEL
LIN {X 0,Y 369.823,Z 705.079,A -85,B 0,C 180,E1 -26449.136,E2 -26449.136} C_VEL
LIN {X 0,Y 379.411,Z 615.126,A -85,B 0,C 180,E1 -26450.408,E2 -26450.408} C_VEL
LIN {X 0,Y 376.924,Z 609.355,A -85,B 0,C 180,E1 -26453.374,E2 -26453.374} C_VEL
LIN {X 0,Y 375.23,Z 605.577,A -85,B 0,C 180,E1 -26456.333,E2 -26456.333} C_VEL
LIN {X 0,Y 374.3,Z 602.133,A -85,B 0,C 180,E1 -26461.225,E2 -26461.225} C_VEL
LIN {X 0,Y 375.612,Z 606.381,A -85,B 0,C 180,E1 -26466.88,E2 -26466.88} C_VEL
LIN {X 0,Y 377.382,Z 610.539,A -85,B 0,C 180,E1 -26469.686,E2 -26469.686} C_VEL
LIN {X 0,Y 379.368,Z 615.06,A -85,B 0,C 180,E1 -26471.968,E2 -26471.968} C_VEL
LIN {X 0,Y 364.694,Z 750.368,A -85,B 0,C 180,E1 -26473.884,E2 -26473.884} C_VEL
LIN {X 0,Y 360.131,Z 776.544,A -85,B 0,C 180,E1 -26474.348,E2 -26474.348} C_VEL
LIN {X 0,Y 355.077,Z 797.804,A -85,B 0,C 180,E1 -26474.834,E2 -26474.834} C_VEL
LIN {X 0,Y 347.273,Z 823.638,A -85,B 0,C 180,E1 -26475.611,E2 -26475.611} C_VEL
LIN {X 0,Y 339.775,Z 843.972,A -85,B 0,C 180,E1 -26476.392,E2 -26476.392} C_VEL
LIN {X 0,Y 329.731,Z 867.163,A -85,B 0,C 180,E1 -26477.503,E2 -26477.503} C_VEL
LIN {X 0,Y 319.79,Z 886.793,A -85,B 0,C 180,E1 -26478.668,E2 -26478.668} C_VEL
LIN {X 0,Y 308.34,Z 906.91,A -85,B 0,C 180,E1 -26480.123,E2 -26480.123} C_VEL
LIN {X 0,Y 295.765,Z 926.18,A -85,B 0,C 180,E1 -26481.875,E2 -26481.875} C_VEL
LIN {X 0,Y 282.715,Z 944.307,A -85,B 0,C 180,E1 -26483.901,E2 -26483.901} C_VEL
LIN {X 0,Y 268.855,Z 961.441,A -85,B 0,C 180,E1 -26486.325,E2 -26486.325} C_VEL
LIN {X 0,Y 255.887,Z 976.185,A -85,B 0,C 180,E1 -26488.921,E2 -26488.921} C_VEL
LIN {X 0,Y 240.634,Z 992.018,A -85,B 0,C 180,E1 -26492.487,E2 -26492.487} C_VEL
LIN {X 0,Y 228.091,Z 1004.089,A -85,B 0,C 180,E1 -26495.975,E2 -26495.975} C_VEL
LIN {X 0,Y 213.113,Z 1017.571,A -85,B 0,C 180,E1 -26501.061,E2 -26501.061} C_VEL
LIN {X 0,Y 201.571,Z 1027.448,A -85,B 0,C 180,E1 -26506.015,E2 -26506.015} C_VEL
LIN {X 0,Y 189.668,Z 1037.363,A -85,B 0,C 180,E1 -26512.681,E2 -26512.681} C_VEL
LIN {X 0,Y 181.615,Z 1044.116,A -85,B 0,C 180,E1 -26518.834,E2 -26518.834} C_VEL
LIN {X 0,Y 174.556,Z 1050.463,A -85,B 0,C 180,E1 -26526.719,E2 -26526.719} C_VEL
LIN {X 0,Y 170.625,Z 1054.488,A -85,B 0,C 180,E1 -26534.013,E2 -26534.013} C_VEL
LIN {X 0,Y 168.685,Z 1057.157,A -85,B 0,C 180,E1 -26541.135,E2 -26541.135} C_VEL
LIN {X 0,Y 168.089,Z 1058.673,A -85,B 0,C 180,E1 -26548.296,E2 -26548.296} C_VEL
LIN {X 0,Y 168.062,Z 1058.969,A -85,B 0,C 180,E1 -26554.778,E2 -26554.778} C_VEL
LIN {X 0,Y 168.488,Z 1058.341,A -85,B 0,C 180,E1 -26561.294,E2 -26561.294} C_VEL
LIN {X 0,Y 170.016,Z 1056.657,A -85,B 0,C 180,E1 -26568.162,E2 -26568.162} C_VEL
LIN {X 0,Y 173.784,Z 1053.449,A -85,B 0,C 180,E1 -26575.93,E2 -26575.93} C_VEL
LIN {X 0,Y 180.307,Z 1048.325,A -85,B 0,C 180,E1 -26583.713,E2 -26583.713} C_VEL
LIN {X 0,Y 188.55,Z 1042.257,A -85,B 0,C 180,E1 -26590.314,E2 -26590.314} C_VEL
LIN {X 0,Y 199.935,Z 1033.803,A -85,B 0,C 180,E1 -26596.9,E2 -26596.9} C_VEL
LIN {X 0,Y 211.107,Z 1025.277,A -85,B 0,C 180,E1 -26601.836,E2 -26601.836} C_VEL
LIN {X 0,Y 226.243,Z 1013.097,A -85,B 0,C 180,E1 -26607.11,E2 -26607.11} C_VEL
LIN {X 0,Y 239.37,Z 1001.756,A -85,B 0,C 180,E1 -26610.813,E2 -26610.813} C_VEL
LIN {X 0,Y 254.891,Z 987.33,A -85,B 0,C 180,E1 -26614.455,E2 -26614.455} C_VEL
LIN {X 0,Y 268.899,Z 972.996,A -85,B 0,C 180,E1 -26617.249,E2 -26617.249} C_VEL
LIN {X 0,Y 283.645,Z 956.609,A -85,B 0,C 180,E1 -26619.79,E2 -26619.79} C_VEL
LIN {X 0,Y 297.668,Z 939.089,A -85,B 0,C 180,E1 -26621.919,E2 -26621.919} C_VEL
LIN {X 0,Y 311.384,Z 920.222,A -85,B 0,C 180,E1 -26623.765,E2 -26623.765} C_VEL
LIN {X 0,Y 324.048,Z 900.26,A -85,B 0,C 180,E1 -26625.317,E2 -26625.317} C_VEL
LIN {X 0,Y 335.603,Z 879.878,A -85,B 0,C 180,E1 -26626.598,E2 -26626.598} C_VEL
LIN {X 0,Y 346.213,Z 857.957,A -85,B 0,C 180,E1 -26627.706,E2 -26627.706} C_VEL
LIN {X 0,Y 354.723,Z 837.755,A -85,B 0,C 180,E1 -26628.531,E2 -26628.531} C_VEL
LIN {X 0,Y 363.018,Z 814.145,A -85,B 0,C 180,E1 -26629.303,E2 -26629.303} C_VEL
LIN {X 0,Y 369.13,Z 792.82,A -85,B 0,C 180,E1 -26629.859,E2 -26629.859} C_VEL
LIN {X 0,Y 375.012,Z 766.175,A -85,B 0,C 180,E1 -26630.382,E2 -26630.382} C_VEL
LIN {X 0,Y 378.442,Z 743.895,A -85,B 0,C 180,E1 -26630.721,E2 -26630.721} C_VEL
LIN {X 0,Y 391.526,Z 625.127,A -85,B 0,C 180,E1 -26632.369,E2 -26632.369} C_VEL
LIN {X 0,Y 390.292,Z 622.227,A -85,B 0,C 180,E1 -26634.118,E2 -26634.118} C_VEL
LIN {X 0,Y 389.23,Z 619.551,A -85,B 0,C 180,E1 -26636.17,E2 -26636.17} C_VEL
LIN {X 0,Y 388.32,Z 616.451,A -85,B 0,C 180,E1 -26641.033,E2 -26641.033} C_VEL
LIN {X 0,Y 389.479,Z 620.134,A -85,B 0,C 180,E1 -26646.042,E2 -26646.042} C_VEL
LIN {X 0,Y 391.107,Z 624.154,A -85,B 0,C 180,E1 -26648.75,E2 -26648.75} C_VEL
LIN {X 0,Y 391.577,Z 625.466,A -85,B 0,C 180,E1 -26649.388,E2 -26649.388} C_VEL
LIN {X 0,Y 383.818,Z 696.159,A -85,B 0,C 180,E1 -26650.345,E2 -26650.345} C_VEL
LIN {X 0,Y 382.804,Z 703.857,A -85,B 0,C 180,E1 -26650.296,E2 -26650.296} C_VEL
LIN {X 0,Y 379.554,Z 724.405,A -85,B 0,C 180,E1 -26649.648,E2 -26649.648} C_VEL
LIN {X 0,Y 378.712,Z 731.006,A -85,B 0,C 180,E1 -26649.627,E2 -26649.627} C_VEL
LIN {X 0,Y 374.403,Z 763.566,A -85,B 0,C 180,E1 -26650.087,E2 -26650.087} C_VEL
LIN {X 0,Y 369.937,Z 785.777,A -85,B 0,C 180,E1 -26650.448,E2 -26650.448} C_VEL
LIN {X 0,Y 363.081,Z 811.326,A -85,B 0,C 180,E1 -26650.954,E2 -26650.954} C_VEL
LIN {X 0,Y 356.554,Z 830.814,A -85,B 0,C 180,E1 -26651.447,E2 -26651.447} C_VEL
LIN {X 0,Y 347.767,Z 853.173,A -85,B 0,C 180,E1 -26652.161,E2 -26652.161} C_VEL
LIN {X 0,Y 337.22,Z 875.538,A -85,B 0,C 180,E1 -26653.085,E2 -26653.085} C_VEL
LIN {X 0,Y 326.794,Z 894.969,A -85,B 0,C 180,E1 -26654.088,E2 -26654.088} C_VEL
LIN {X 0,Y 313.803,Z 916.07,A -85,B 0,C 180,E1 -26655.447,E2 -26655.447} C_VEL
LIN {X 0,Y 301.891,Z 933.296,A -85,B 0,C 180,E1 -26656.825,E2 -26656.825} C_VEL
LIN {X 0,Y 286.342,Z 953.416,A -85,B 0,C 180,E1 -26658.859,E2 -26658.859} C_VEL
LIN {X 0,Y 272.86,Z 969.042,A -85,B 0,C 180,E1 -26660.862,E2 -26660.862} C_VEL
LIN {X 0,Y 257.362,Z 985.48,A -85,B 0,C 180,E1 -26663.524,E2 -26663.524} C_VEL
LIN {X 0,Y 242.492,Z 999.713,A -85,B 0,C 180,E1 -26666.52,E2 -26666.52} C_VEL
LIN {X 0,Y 226.954,Z 1013.579,A -85,B 0,C 180,E1 -26670.286,E2 -26670.286} C_VEL
LIN {X 0,Y 211.85,Z 1025.867,A -85,B 0,C 180,E1 -26674.79,E2 -26674.79} C_VEL
LIN {X 0,Y 198.226,Z 1036.496,A -85,B 0,C 180,E1 -26679.94,E2 -26679.94} C_VEL
LIN {X 0,Y 185.84,Z 1045.617,A -85,B 0,C 180,E1 -26686.047,E2 -26686.047} C_VEL
LIN {X 0,Y 175.868,Z 1053.025,A -85,B 0,C 180,E1 -26692.747,E2 -26692.747} C_VEL
LIN {X 0,Y 167.748,Z 1059.227,A -85,B 0,C 180,E1 -26700.74,E2 -26700.74} C_VEL
LIN {X 0,Y 163.166,Z 1063.196,A -85,B 0,C 180,E1 -26708.049,E2 -26708.049} C_VEL
LIN {X 0,Y 160.515,Z 1066.259,A -85,B 0,C 180,E1 -26716.674,E2 -26716.674} C_VEL
LIN {X 0,Y 159.993,Z 1067.511,A -85,B 0,C 180,E1 -26724.261,E2 -26724.261} C_VEL
LIN {X 0,Y 160.051,Z 1067.671,A -85,B 0,C 180,E1 -26730,E2 -26730} C_VEL
LIN {X 0,Y 159.998,Z 1067.089,A -85,B 0,C 180,E1 -26735.739,E2 -26735.739} C_VEL
LIN {X 0,Y 160.393,Z 1065.414,A -85,B 0,C 180,E1 -26742.603,E2 -26742.603} C_VEL
LIN {X 0,Y 162.21,Z 1062.558,A -85,B 0,C 180,E1 -26749.818,E2 -26749.818} C_VEL
LIN {X 0,Y 167.087,Z 1057.38,A -85,B 0,C 180,E1 -26758.603,E2 -26758.603} C_VEL
LIN {X 0,Y 173.95,Z 1051.191,A -85,B 0,C 180,E1 -26765.896,E2 -26765.896} C_VEL
LIN {X 0,Y 184.077,Z 1042.81,A -85,B 0,C 180,E1 -26773.19,E2 -26773.19} C_VEL
LIN {X 0,Y 195.529,Z 1033.277,A -85,B 0,C 180,E1 -26779.186,E2 -26779.186} C_VEL
LIN {X 0,Y 208.793,Z 1022.136,A -85,B 0,C 180,E1 -26784.5,E2 -26784.5} C_VEL
LIN {X 0,Y 222.871,Z 1009.473,A -85,B 0,C 180,E1 -26788.971,E2 -26788.971} C_VEL
LIN {X 0,Y 237.376,Z 995.722,A -85,B 0,C 180,E1 -26792.721,E2 -26792.721} C_VEL
LIN {X 0,Y 251.975,Z 980.561,A -85,B 0,C 180,E1 -26795.879,E2 -26795.879} C_VEL
LIN {X 0,Y 265.626,Z 965.239,A -85,B 0,C 180,E1 -26798.4,E2 -26798.4} C_VEL
LIN {X 0,Y 281.011,Z 946.124,A -85,B 0,C 180,E1 -26800.856,E2 -26800.856} C_VEL
LIN {X 0,Y 293.403,Z 929.045,A -85,B 0,C 180,E1 -26802.595,E2 -26802.595} C_VEL
LIN {X 0,Y 307.394,Z 907.422,A -85,B 0,C 180,E1 -26804.337,E2 -26804.337} C_VEL
LIN {X 0,Y 318.047,Z 888.773,A -85,B 0,C 180,E1 -26805.535,E2 -26805.535} C_VEL
LIN {X 0,Y 329.303,Z 866.351,A -85,B 0,C 180,E1 -26806.695,E2 -26806.695} C_VEL
LIN {X 0,Y 338.031,Z 846.016,A -85,B 0,C 180,E1 -26807.53,E2 -26807.53} C_VEL
LIN {X 0,Y 346.679,Z 822.568,A -85,B 0,C 180,E1 -26808.289,E2 -26808.289} C_VEL
LIN {X 0,Y 353.619,Z 798.987,A -85,B 0,C 180,E1 -26808.864,E2 -26808.864} C_VEL
LIN {X 0,Y 359.328,Z 774.575,A -85,B 0,C 180,E1 -26809.331,E2 -26809.331} C_VEL
LIN {X 0,Y 363.205,Z 750.195,A -85,B 0,C 180,E1 -26809.72,E2 -26809.72} C_VEL
LIN {X 0,Y 377.338,Z 620.996,A -85,B 0,C 180,E1 -26811.535,E2 -26811.535} C_VEL
LIN {X 0,Y 375.456,Z 616.572,A -85,B 0,C 180,E1 -26814.038,E2 -26814.038} C_VEL
LIN {X 0,Y 374.181,Z 613.455,A -85,B 0,C 180,E1 -26816.476,E2 -26816.476} C_VEL
LIN {X 0,Y 373.307,Z 610.23,A -85,B 0,C 180,E1 -26821.381,E2 -26821.381} C_VEL
LIN {X 0,Y 374.514,Z 614.191,A -85,B 0,C 180,E1 -26826.669,E2 -26826.669} C_VEL
LIN {X 0,Y 376.161,Z 618.235,A -85,B 0,C 180,E1 -26829.409,E2 -26829.409} C_VEL
LIN {X 0,Y 377.304,Z 621.025,A -85,B 0,C 180,E1 -26830.855,E2 -26830.855} C_VEL
LIN {X 0,Y 362.994,Z 750.615,A -85,B 0,C 180,E1 -26832.652,E2 -26832.652} C_VEL
LIN {X 0,Y 358.383,Z 776.712,A -85,B 0,C 180,E1 -26833.101,E2 -26833.101} C_VEL
LIN {X 0,Y 353.225,Z 798.122,A -85,B 0,C 180,E1 -26833.574,E2 -26833.574} C_VEL
LIN {X 0,Y 345.66,Z 822.949,A -85,B 0,C 180,E1 -26834.291,E2 -26834.291} C_VEL
LIN {X 0,Y 338.053,Z 843.393,A -85,B 0,C 180,E1 -26835.046,E2 -26835.046} C_VEL
LIN {X 0,Y 328.741,Z 864.964,A -85,B 0,C 180,E1 -26836.026,E2 -26836.026} C_VEL
LIN {X 0,Y 318.186,Z 885.639,A -85,B 0,C 180,E1 -26837.194,E2 -26837.194} C_VEL
LIN {X 0,Y 306.908,Z 905.258,A -85,B 0,C 180,E1 -26838.547,E2 -26838.547} C_VEL
LIN {X 0,Y 293.697,Z 925.372,A -85,B 0,C 180,E1 -26840.292,E2 -26840.292} C_VEL
LIN {X 0,Y 281.589,Z 941.945,A -85,B 0,C 180,E1 -26842.062,E2 -26842.062} C_VEL
LIN {X 0,Y 266.157,Z 960.88,A -85,B 0,C 180,E1 -26844.614,E2 -26844.614} C_VEL
LIN {X 0,Y 252.825,Z 975.694,A -85,B 0,C 180,E1 -26847.146,E2 -26847.146} C_VEL
LIN {X 0,Y 236.713,Z 992.009,A -85,B 0,C 180,E1 -26850.738,E2 -26850.738} C_VEL
LIN {X 0,Y 223.669,Z 1004.158,A -85,B 0,C 180,E1 -26854.206,E2 -26854.206} C_VEL
LIN {X 0,Y 208.646,Z 1017.213,A -85,B 0,C 180,E1 -26859.073,E2 -26859.073} C_VEL
LIN {X 0,Y 196.884,Z 1026.835,A -85,B 0,C 180,E1 -26863.85,E2 -26863.85} C_VEL
LIN {X 0,Y 185.094,Z 1036.253,A -85,B 0,C 180,E1 -26869.996,E2 -26869.996} C_VEL
LIN {X 0,Y 175.429,Z 1043.788,A -85,B 0,C 180,E1 -26876.827,E2 -26876.827} C_VEL
LIN {X 0,Y 167.887,Z 1050.102,A -85,B 0,C 180,E1 -26884.608,E2 -26884.608} C_VEL
LIN {X 0,Y 163.02,Z 1054.573,A -85,B 0,C 180,E1 -26892.878,E2 -26892.878} C_VEL
LIN {X 0,Y 160.88,Z 1057.168,A -85,B 0,C 180,E1 -26899.978,E2 -26899.978} C_VEL
LIN {X 0,Y 160.109,Z 1058.838,A -85,B 0,C 180,E1 -26907.733,E2 -26907.733} C_VEL
LIN {X 0,Y 160.056,Z 1059.223,A -85,B 0,C 180,E1 -26914.299,E2 -26914.299} C_VEL
LIN {X 0,Y 160.511,Z 1058.611,A -85,B 0,C 180,E1 -26921.499,E2 -26921.499} C_VEL
LIN {X 0,Y 162.153,Z 1056.967,A -85,B 0,C 180,E1 -26928.702,E2 -26928.702} C_VEL
LIN {X 0,Y 165.963,Z 1053.953,A -85,B 0,C 180,E1 -26936.477,E2 -26936.477} C_VEL
LIN {X 0,Y 173.154,Z 1048.748,A -85,B 0,C 180,E1 -26944.916,E2 -26944.916} C_VEL
LIN {X 0,Y 181.86,Z 1042.73,A -85,B 0,C 180,E1 -26951.703,E2 -26951.703} C_VEL
LIN {X 0,Y 194.363,Z 1033.962,A -85,B 0,C 180,E1 -26958.685,E2 -26958.685} C_VEL
LIN {X 0,Y 206.413,Z 1025.189,A -85,B 0,C 180,E1 -26963.773,E2 -26963.773} C_VEL
LIN {X 0,Y 221.852,Z 1013.231,A -85,B 0,C 180,E1 -26968.907,E2 -26968.907} C_VEL
LIN {X 0,Y 235.447,Z 1001.881,A -85,B 0,C 180,E1 -26972.57,E2 -26972.57} C_VEL
LIN {X 0,Y 251.444,Z 987.434,A -85,B 0,C 180,E1 -26976.151,E2 -26976.151} C_VEL
LIN {X 0,Y 265.821,Z 973.094,A -85,B 0,C 180,E1 -26978.885,E2 -26978.885} C_VEL
LIN {X 0,Y 281.159,Z 956.384,A -85,B 0,C 180,E1 -26981.398,E2 -26981.398} C_VEL
LIN {X 0,Y 294.798,Z 939.696,A -85,B 0,C 180,E1 -26983.371,E2 -26983.371} C_VEL
LIN {X 0,Y 308.318,Z 921.484,A -85,B 0,C 180,E1 -26985.112,E2 -26985.112} C_VEL
LIN {X 0,Y 321.185,Z 901.731,A -85,B 0,C 180,E1 -26986.619,E2 -26986.619} C_VEL
LIN {X 0,Y 331.998,Z 883.105,A -85,B 0,C 180,E1 -26987.771,E2 -26987.771} C_VEL
LIN {X 0,Y 343.585,Z 860.065,A -85,B 0,C 180,E1 -26988.926,E2 -26988.926} C_VEL
LIN {X 0,Y 352.069,Z 840.421,A -85,B 0,C 180,E1 -26989.715,E2 -26989.715} C_VEL
LIN {X 0,Y 360.678,Z 816.897,A -85,B 0,C 180,E1 -26990.48,E2 -26990.48} C_VEL
LIN {X 0,Y 367.215,Z 794.695,A -85,B 0,C 180,E1 -26991.047,E2 -26991.047} C_VEL
LIN {X 0,Y 372.937,Z 770.193,A -85,B 0,C 180,E1 -26991.527,E2 -26991.527} C_VEL
LIN {X 0,Y 376.783,Z 746.415,A -85,B 0,C 180,E1 -26991.885,E2 -26991.885} C_VEL
LIN {X 0,Y 389.739,Z 631.344,A -85,B 0,C 180,E1 -26993.437,E2 -26993.437} C_VEL
LIN {X 0,Y 388.184,Z 627.432,A -85,B 0,C 180,E1 -26996.308,E2 -26996.308} C_VEL
LIN {X 0,Y 387.351,Z 624.331,A -85,B 0,C 180,E1 -27000.887,E2 -27000.887} C_VEL
LIN {X 0,Y 388.422,Z 628.053,A -85,B 0,C 180,E1 -27005.91,E2 -27005.91} C_VEL
LIN {X 0,Y 389.773,Z 631.614,A -85,B 0,C 180,E1 -27008.306,E2 -27008.306} C_VEL
LIN {X 0,Y 378.712,Z 731.006,A -85,B 0,C 180,E1 -27009.627,E2 -27009.627} C_VEL
LIN {X 0,Y 377.714,Z 738.7,A -85,B 0,C 180,E1 -27009.58,E2 -27009.58} C_VEL
LIN {X 0,Y 374.068,Z 759.174,A -85,B 0,C 180,E1 -27008.908,E2 -27008.908} C_VEL
LIN {X 0,Y 372.792,Z 765.719,A -85,B 0,C 180,E1 -27008.904,E2 -27008.904} C_VEL
LIN {X 0,Y 367.836,Z 789.395,A -85,B 0,C 180,E1 -27009.279,E2 -27009.279} C_VEL
LIN {X 0,Y 361.168,Z 813.019,A -85,B 0,C 180,E1 -27009.741,E2 -27009.741} C_VEL
LIN {X 0,Y 354.164,Z 833.38,A -85,B 0,C 180,E1 -27010.245,E2 -27010.245} C_VEL
LIN {X 0,Y 344.297,Z 857.319,A -85,B 0,C 180,E1 -27011.008,E2 -27011.008} C_VEL
LIN {X 0,Y 334.562,Z 877.375,A -85,B 0,C 180,E1 -27011.824,E2 -27011.824} C_VEL
LIN {X 0,Y 322.636,Z 898.882,A -85,B 0,C 180,E1 -27012.922,E2 -27012.922} C_VEL
LIN {X 0,Y 310.386,Z 918.046,A -85,B 0,C 180,E1 -27014.151,E2 -27014.151} C_VEL
LIN {X 0,Y 296.979,Z 936.905,A -85,B 0,C 180,E1 -27015.65,E2 -27015.65} C_VEL
LIN {X 0,Y 282.07,Z 955.374,A -85,B 0,C 180,E1 -27017.53,E2 -27017.53} C_VEL
LIN {X 0,Y 268.359,Z 970.812,A -85,B 0,C 180,E1 -27019.496,E2 -27019.496} C_VEL
LIN {X 0,Y 251.739,Z 987.693,A -85,B 0,C 180,E1 -27022.262,E2 -27022.262} C_VEL
LIN {X 0,Y 237.36,Z 1001.003,A -85,B 0,C 180,E1 -27025.083,E2 -27025.083} C_VEL
LIN {X 0,Y 219.956,Z 1015.757,A -85,B 0,C 180,E1 -27029.214,E2 -27029.214} C_VEL
LIN {X 0,Y 205.881,Z 1026.76,A -85,B 0,C 180,E1 -27033.348,E2 -27033.348} C_VEL
LIN {X 0,Y 190.594,Z 1038.003,A -85,B 0,C 180,E1 -27039.065,E2 -27039.065} C_VEL
LIN {X 0,Y 178.933,Z 1046.164,A -85,B 0,C 180,E1 -27044.791,E2 -27044.791} C_VEL
LIN {X 0,Y 167.932,Z 1053.856,A -85,B 0,C 180,E1 -27052.173,E2 -27052.173} C_VEL
LIN {X 0,Y 160.029,Z 1059.461,A -85,B 0,C 180,E1 -27060.009,E2 -27060.009} C_VEL
LIN {X 0,Y 154.899,Z 1063.661,A -85,B 0,C 180,E1 -27068.411,E2 -27068.411} C_VEL
LIN {X 0,Y 152.378,Z 1066.343,A -85,B 0,C 180,E1 -27077.494,E2 -27077.494} C_VEL
LIN {X 0,Y 151.995,Z 1067.325,A -85,B 0,C 180,E1 -27084.337,E2 -27084.337} C_VEL
LIN {X 0,Y 152.054,Z 1067.454,A -85,B 0,C 180,E1 -27090,E2 -27090} C_VEL
LIN {X 0,Y 151.999,Z 1066.865,A -85,B 0,C 180,E1 -27096.042,E2 -27096.042} C_VEL
LIN {X 0,Y 152.481,Z 1065.182,A -85,B 0,C 180,E1 -27103.268,E2 -27103.268} C_VEL
LIN {X 0,Y 154.529,Z 1062.318,A -85,B 0,C 180,E1 -27110.847,E2 -27110.847} C_VEL
LIN {X 0,Y 159.895,Z 1057.125,A -85,B 0,C 180,E1 -27120.018,E2 -27120.018} C_VEL
LIN {X 0,Y 167.312,Z 1050.928,A -85,B 0,C 180,E1 -27127.559,E2 -27127.559} C_VEL
LIN {X 0,Y 178.116,Z 1042.531,A -85,B 0,C 180,E1 -27135.018,E2 -27135.018} C_VEL
LIN {X 0,Y 190.201,Z 1032.991,A -85,B 0,C 180,E1 -27141.081,E2 -27141.081} C_VEL
LIN {X 0,Y 204.082,Z 1021.838,A -85,B 0,C 180,E1 -27146.398,E2 -27146.398} C_VEL
LIN {X 0,Y 218.709,Z 1009.161,A -85,B 0,C 180,E1 -27150.834,E2 -27150.834} C_VEL
LIN {X 0,Y 233.696,Z 995.401,A -85,B 0,C 180,E1 -27154.526,E2 -27154.526} C_VEL
LIN {X 0,Y 248.713,Z 980.22,A -85,B 0,C 180,E1 -27157.617,E2 -27157.617} C_VEL
LIN {X 0,Y 262.703,Z 964.888,A -85,B 0,C 180,E1 -27160.072,E2 -27160.072} C_VEL
LIN {X 0,Y 278.275,Z 945.943,A -85,B 0,C 180,E1 -27162.433,E2 -27162.433} C_VEL
LIN {X 0,Y 290.616,Z 929.27,A -85,B 0,C 180,E1 -27164.08,E2 -27164.08} C_VEL
LIN {X 0,Y 304.787,Z 907.829,A -85,B 0,C 180,E1 -27165.756,E2 -27165.756} C_VEL
LIN {X 0,Y 315.652,Z 889.153,A -85,B 0,C 180,E1 -27166.919,E2 -27166.919} C_VEL
LIN {X 0,Y 326.777,Z 867.511,A -85,B 0,C 180,E1 -27168.007,E2 -27168.007} C_VEL
LIN {X 0,Y 336.035,Z 846.315,A -85,B 0,C 180,E1 -27168.848,E2 -27168.848} C_VEL
LIN {X 0,Y 344.662,Z 823.368,A -85,B 0,C 180,E1 -27169.566,E2 -27169.566} C_VEL
LIN {X 0,Y 351.856,Z 799.376,A -85,B 0,C 180,E1 -27170.131,E2 -27170.131} C_VEL
LIN {X 0,Y 357.615,Z 775.258,A -85,B 0,C 180,E1 -27170.576,E2 -27170.576} C_VEL
LIN {X 0,Y 361.655,Z 750.471,A -85,B 0,C 180,E1 -27170.96,E2 -27170.96} C_VEL
LIN {X 0,Y 375.403,Z 627.088,A -85,B 0,C 180,E1 -27172.655,E2 -27172.655} C_VEL
LIN {X 0,Y 374.084,Z 623.885,A -85,B 0,C 180,E1 -27174.632,E2 -27174.632} C_VEL
LIN {X 0,Y 373.134,Z 621.334,A -85,B 0,C 180,E1 -27176.62,E2 -27176.62} C_VEL
LIN {X 0,Y 372.326,Z 618.216,A -85,B 0,C 180,E1 -27181.385,E2 -27181.385} C_VEL
LIN {X 0,Y 373.453,Z 622.113,A -85,B 0,C 180,E1 -27186.534,E2 -27186.534} C_VEL
LIN {X 0,Y 374.948,Z 625.93,A -85,B 0,C 180,E1 -27189.13,E2 -27189.13} C_VEL
LIN {X 0,Y 375.361,Z 627.187,A -85,B 0,C 180,E1 -27189.732,E2 -27189.732} C_VEL
LIN {X 0,Y 361.464,Z 750.862,A -85,B 0,C 180,E1 -27191.41,E2 -27191.41} C_VEL
LIN {X 0,Y 356.777,Z 777.011,A -85,B 0,C 180,E1 -27191.845,E2 -27191.845} C_VEL
LIN {X 0,Y 351.552,Z 798.416,A -85,B 0,C 180,E1 -27192.301,E2 -27192.301} C_VEL
LIN {X 0,Y 343.776,Z 823.534,A -85,B 0,C 180,E1 -27193.002,E2 -27193.002} C_VEL
LIN {X 0,Y 336.068,Z 843.934,A -85,B 0,C 180,E1 -27193.731,E2 -27193.731} C_VEL
LIN {X 0,Y 326.126,Z 866.42,A -85,B 0,C 180,E1 -27194.725,E2 -27194.725} C_VEL
LIN {X 0,Y 315.463,Z 886.892,A -85,B 0,C 180,E1 -27195.852,E2 -27195.852} C_VEL
LIN {X 0,Y 303.574,Z 907.129,A -85,B 0,C 180,E1 -27197.219,E2 -27197.219} C_VEL
LIN {X 0,Y 290.382,Z 926.631,A -85,B 0,C 180,E1 -27198.886,E2 -27198.886} C_VEL
LIN {X 0,Y 276.56,Z 945.065,A -85,B 0,C 180,E1 -27200.837,E2 -27200.837} C_VEL
LIN {X 0,Y 262.07,Z 962.147,A -85,B 0,C 180,E1 -27203.147,E2 -27203.147} C_VEL
LIN {X 0,Y 248.439,Z 976.868,A -85,B 0,C 180,E1 -27205.64,E2 -27205.64} C_VEL
LIN {X 0,Y 232.261,Z 992.697,A -85,B 0,C 180,E1 -27209.109,E2 -27209.109} C_VEL
LIN {X 0,Y 218.488,Z 1005.095,A -85,B 0,C 180,E1 -27212.642,E2 -27212.642} C_VEL
LIN {X 0,Y 202.958,Z 1018.013,A -85,B 0,C 180,E1 -27217.516,E2 -27217.516} C_VEL
LIN {X 0,Y 190.742,Z 1027.571,A -85,B 0,C 180,E1 -27222.342,E2 -27222.342} C_VEL
LIN {X 0,Y 177.939,Z 1037.213,A -85,B 0,C 180,E1 -27228.894,E2 -27228.894} C_VEL
LIN {X 0,Y 168.28,Z 1044.346,A -85,B 0,C 180,E1 -27235.634,E2 -27235.634} C_VEL
LIN {X 0,Y 160.311,Z 1050.558,A -85,B 0,C 180,E1 -27243.715,E2 -27243.715} C_VEL
LIN {X 0,Y 155.313,Z 1054.813,A -85,B 0,C 180,E1 -27252,E2 -27252} C_VEL
LIN {X 0,Y 152.896,Z 1057.51,A -85,B 0,C 180,E1 -27259.83,E2 -27259.83} C_VEL
LIN {X 0,Y 152.112,Z 1059.078,A -85,B 0,C 180,E1 -27267.74,E2 -27267.74} C_VEL
LIN {X 0,Y 152.062,Z 1059.433,A -85,B 0,C 180,E1 -27274.526,E2 -27274.526} C_VEL
LIN {X 0,Y 152.585,Z 1058.817,A -85,B 0,C 180,E1 -27282.105,E2 -27282.105} C_VEL
LIN {X 0,Y 154.442,Z 1057.168,A -85,B 0,C 180,E1 -27289.673,E2 -27289.673} C_VEL
LIN {X 0,Y 158.647,Z 1054.149,A -85,B 0,C 180,E1 -27297.8,E2 -27297.8} C_VEL
LIN {X 0,Y 166.393,Z 1048.96,A -85,B 0,C 180,E1 -27306.506,E2 -27306.506} C_VEL
LIN {X 0,Y 175.285,Z 1043.202,A -85,B 0,C 180,E1 -27313.198,E2 -27313.198} C_VEL
LIN {X 0,Y 188.413,Z 1034.522,A -85,B 0,C 180,E1 -27320.309,E2 -27320.309} C_VEL
LIN {X 0,Y 201.002,Z 1025.774,A -85,B 0,C 180,E1 -27325.452,E2 -27325.452} C_VEL
LIN {X 0,Y 216.974,Z 1013.934,A -85,B 0,C 180,E1 -27330.572,E2 -27330.572} C_VEL
LIN {X 0,Y 230.992,Z 1002.637,A -85,B 0,C 180,E1 -27334.206,E2 -27334.206} C_VEL
LIN {X 0,Y 246.815,Z 988.886,A -85,B 0,C 180,E1 -27337.616,E2 -27337.616} C_VEL
LIN {X 0,Y 262.135,Z 974.029,A -85,B 0,C 180,E1 -27340.417,E2 -27340.417} C_VEL
LIN {X 0,Y 277.791,Z 957.455,A -85,B 0,C 180,E1 -27342.872,E2 -27342.872} C_VEL
LIN {X 0,Y 292.122,Z 940.304,A -85,B 0,C 180,E1 -27344.85,E2 -27344.85} C_VEL
LIN {X 0,Y 305.426,Z 922.738,A -85,B 0,C 180,E1 -27346.485,E2 -27346.485} C_VEL
LIN {X 0,Y 318.945,Z 902.467,A -85,B 0,C 180,E1 -27347.992,E2 -27347.992} C_VEL
LIN {X 0,Y 329.913,Z 883.896,A -85,B 0,C 180,E1 -27349.103,E2 -27349.103} C_VEL
LIN {X 0,Y 341.912,Z 860.439,A -85,B 0,C 180,E1 -27350.24,E2 -27350.24} C_VEL
LIN {X 0,Y 350.295,Z 841.325,A -85,B 0,C 180,E1 -27350.979,E2 -27350.979} C_VEL
LIN {X 0,Y 358.981,Z 818.101,A -85,B 0,C 180,E1 -27351.712,E2 -27351.712} C_VEL
LIN {X 0,Y 365.752,Z 795.493,A -85,B 0,C 180,E1 -27352.271,E2 -27352.271} C_VEL
LIN {X 0,Y 371.546,Z 771.253,A -85,B 0,C 180,E1 -27352.731,E2 -27352.731} C_VEL
LIN {X 0,Y 375.564,Z 746.851,A -85,B 0,C 180,E1 -27353.087,E2 -27353.087} C_VEL
LIN {X 0,Y 388.046,Z 637.82,A -85,B 0,C 180,E1 -27354.529,E2 -27354.529} C_VEL
LIN {X 0,Y 387.076,Z 635.217,A -85,B 0,C 180,E1 -27356.594,E2 -27356.594} C_VEL
LIN {X 0,Y 386.369,Z 632.327,A -85,B 0,C 180,E1 -27360.89,E2 -27360.89} C_VEL
LIN {X 0,Y 387.338,Z 635.859,A -85,B 0,C 180,E1 -27365.704,E2 -27365.704} C_VEL
LIN {X 0,Y 388.067,Z 638.147,A -85,B 0,C 180,E1 -27367.217,E2 -27367.217} C_VEL
LIN {X 0,Y 374.709,Z 754.049,A -85,B 0,C 180,E1 -27368.735,E2 -27368.735} C_VEL
LIN {X 0,Y 372.792,Z 765.719,A -85,B 0,C 180,E1 -27368.904,E2 -27368.904} C_VEL
LIN {X 0,Y 371.277,Z 773.317,A -85,B 0,C 180,E1 -27368.847,E2 -27368.847} C_VEL
LIN {X 0,Y 365.768,Z 793.421,A -85,B 0,C 180,E1 -27368.2,E2 -27368.2} C_VEL
LIN {X 0,Y 363.895,Z 799.826,A -85,B 0,C 180,E1 -27368.218,E2 -27368.218} C_VEL
LIN {X 0,Y 356.423,Z 823.805,A -85,B 0,C 180,E1 -27368.713,E2 -27368.713} C_VEL
LIN {X 0,Y 348.041,Z 845.479,A -85,B 0,C 180,E1 -27369.305,E2 -27369.305} C_VEL
LIN {X 0,Y 338.627,Z 866.422,A -85,B 0,C 180,E1 -27370.02,E2 -27370.02} C_VEL
LIN {X 0,Y 326.946,Z 888.501,A -85,B 0,C 180,E1 -27370.977,E2 -27370.977} C_VEL
LIN {X 0,Y 315.383,Z 907.692,A -85,B 0,C 180,E1 -27372.022,E2 -27372.022} C_VEL
LIN {X 0,Y 300.755,Z 928.939,A -85,B 0,C 180,E1 -27373.481,E2 -27373.481} C_VEL
LIN {X 0,Y 287.707,Z 945.803,A -85,B 0,C 180,E1 -27374.95,E2 -27374.95} C_VEL
LIN {X 0,Y 270.941,Z 965.149,A -85,B 0,C 180,E1 -27377.094,E2 -27377.094} C_VEL
LIN {X 0,Y 256.316,Z 980.279,A -85,B 0,C 180,E1 -27379.258,E2 -27379.258} C_VEL
LIN {X 0,Y 238.838,Z 996.651,A -85,B 0,C 180,E1 -27382.3,E2 -27382.3} C_VEL
LIN {X 0,Y 223.7,Z 1009.49,A -85,B 0,C 180,E1 -27385.459,E2 -27385.459} C_VEL
LIN {X 0,Y 207.161,Z 1022.449,A -85,B 0,C 180,E1 -27389.681,E2 -27389.681} C_VEL
LIN {X 0,Y 192.57,Z 1032.93,A -85,B 0,C 180,E1 -27394.352,E2 -27394.352} C_VEL
LIN {X 0,Y 178.251,Z 1042.757,A -85,B 0,C 180,E1 -27400.281,E2 -27400.281} C_VEL
LIN {X 0,Y 166.033,Z 1050.649,A -85,B 0,C 180,E1 -27407.116,E2 -27407.116} C_VEL
LIN {X 0,Y 156.312,Z 1057.058,A -85,B 0,C 180,E1 -27414.851,E2 -27414.851} C_VEL
LIN {X 0,Y 148.961,Z 1062.123,A -85,B 0,C 180,E1 -27424.088,E2 -27424.088} C_VEL
LIN {X 0,Y 145.407,Z 1065.091,A -85,B 0,C 180,E1 -27432.388,E2 -27432.388} C_VEL
LIN {X 0,Y 144.033,Z 1066.956,A -85,B 0,C 180,E1 -27441.617,E2 -27441.617} C_VEL
LIN {X 0,Y 144.033,Z 1067.319,A -85,B 0,C 180,E1 -27448.518,E2 -27448.518} C_VEL
LIN {X 0,Y 144.001,Z 1066.922,A -85,B 0,C 180,E1 -27454.78,E2 -27454.78} C_VEL
LIN {X 0,Y 144.399,Z 1065.305,A -85,B 0,C 180,E1 -27462.802,E2 -27462.802} C_VEL
LIN {X 0,Y 146.424,Z 1062.574,A -85,B 0,C 180,E1 -27470.799,E2 -27470.799} C_VEL
LIN {X 0,Y 151.07,Z 1058.295,A -85,B 0,C 180,E1 -27479.326,E2 -27479.326} C_VEL
LIN {X 0,Y 159.581,Z 1051.598,A -85,B 0,C 180,E1 -27488.338,E2 -27488.338} C_VEL
LIN {X 0,Y 169.211,Z 1044.499,A -85,B 0,C 180,E1 -27495.161,E2 -27495.161} C_VEL
LIN {X 0,Y 183.245,Z 1034.109,A -85,B 0,C 180,E1 -27502.298,E2 -27502.298} C_VEL
LIN {X 0,Y 196.167,Z 1024.178,A -85,B 0,C 180,E1 -27507.249,E2 -27507.249} C_VEL
LIN {X 0,Y 213.075,Z 1010.331,A -85,B 0,C 180,E1 -27512.317,E2 -27512.317} C_VEL
LIN {X 0,Y 227.093,Z 997.928,A -85,B 0,C 180,E1 -27515.702,E2 -27515.702} C_VEL
LIN {X 0,Y 244.223,Z 981.397,A -85,B 0,C 180,E1 -27519.133,E2 -27519.133} C_VEL
LIN {X 0,Y 258.302,Z 966.413,A -85,B 0,C 180,E1 -27521.513,E2 -27521.513} C_VEL
LIN {X 0,Y 273.869,Z 948.18,A -85,B 0,C 180,E1 -27523.782,E2 -27523.782} C_VEL
LIN {X 0,Y 287.136,Z 930.725,A -85,B 0,C 180,E1 -27525.484,E2 -27525.484} C_VEL
LIN {X 0,Y 300.657,Z 911.038,A -85,B 0,C 180,E1 -27527.014,E2 -27527.014} C_VEL
LIN {X 0,Y 312.993,Z 890.336,A -85,B 0,C 180,E1 -27528.278,E2 -27528.278} C_VEL
LIN {X 0,Y 323.623,Z 870.228,A -85,B 0,C 180,E1 -27529.27,E2 -27529.27} C_VEL
LIN {X 0,Y 333.881,Z 847.437,A -85,B 0,C 180,E1 -27530.154,E2 -27530.154} C_VEL
LIN {X 0,Y 341.873,Z 826.674,A -85,B 0,C 180,E1 -27530.786,E2 -27530.786} C_VEL
LIN {X 0,Y 349.827,Z 801.391,A -85,B 0,C 180,E1 -27531.376,E2 -27531.376} C_VEL
LIN {X 0,Y 355.241,Z 779.522,A -85,B 0,C 180,E1 -27531.771,E2 -27531.771} C_VEL
LIN {X 0,Y 360.011,Z 752.727,A -85,B 0,C 180,E1 -27532.183,E2 -27532.183} C_VEL
LIN {X 0,Y 373.612,Z 633.289,A -85,B 0,C 180,E1 -27533.77,E2 -27533.77} C_VEL
LIN {X 0,Y 372.089,Z 629.213,A -85,B 0,C 180,E1 -27536.765,E2 -27536.765} C_VEL
LIN {X 0,Y 371.346,Z 626.202,A -85,B 0,C 180,E1 -27541.389,E2 -27541.389} C_VEL
LIN {X 0,Y 372.364,Z 629.922,A -85,B 0,C 180,E1 -27546.321,E2 -27546.321} C_VEL
LIN {X 0,Y 373.577,Z 633.217,A -85,B 0,C 180,E1 -27548.596,E2 -27548.596} C_VEL
LIN {X 0,Y 360.091,Z 751.213,A -85,B 0,C 180,E1 -27550.16,E2 -27550.16} C_VEL
LIN {X 0,Y 355.373,Z 777.18,A -85,B 0,C 180,E1 -27550.576,E2 -27550.576} C_VEL
LIN {X 0,Y 350.07,Z 798.648,A -85,B 0,C 180,E1 -27551.015,E2 -27551.015} C_VEL
LIN {X 0,Y 342.069,Z 824.118,A -85,B 0,C 180,E1 -27551.699,E2 -27551.699} C_VEL
LIN {X 0,Y 334.261,Z 844.475,A -85,B 0,C 180,E1 -27552.4,E2 -27552.4} C_VEL
LIN {X 0,Y 324.182,Z 866.895,A -85,B 0,C 180,E1 -27553.355,E2 -27553.355} C_VEL
LIN {X 0,Y 313.817,Z 886.539,A -85,B 0,C 180,E1 -27554.394,E2 -27554.394} C_VEL
LIN {X 0,Y 301.733,Z 906.842,A -85,B 0,C 180,E1 -27555.706,E2 -27555.706} C_VEL
LIN {X 0,Y 288.501,Z 926.158,A -85,B 0,C 180,E1 -27557.287,E2 -27557.287} C_VEL
LIN {X 0,Y 275.499,Z 943.251,A -85,B 0,C 180,E1 -27559.012,E2 -27559.012} C_VEL
LIN {X 0,Y 259.827,Z 961.586,A -85,B 0,C 180,E1 -27561.364,E2 -27561.364} C_VEL
LIN {X 0,Y 245.843,Z 976.377,A -85,B 0,C 180,E1 -27563.778,E2 -27563.778} C_VEL
LIN {X 0,Y 229.224,Z 992.292,A -85,B 0,C 180,E1 -27567.145,E2 -27567.145} C_VEL
LIN {X 0,Y 215.661,Z 1004.157,A -85,B 0,C 180,E1 -27570.417,E2 -27570.417} C_VEL
LIN {X 0,Y 200.122,Z 1016.792,A -85,B 0,C 180,E1 -27574.974,E2 -27574.974} C_VEL
LIN {X 0,Y 186.559,Z 1026.959,A -85,B 0,C 180,E1 -27579.966,E2 -27579.966} C_VEL
